(* IEC 61131-3 sources: F100R_S278_Temperville/MyController.device.xml.v3^/Plc Logic.plclogic.xml.v3^/Application.application.xml.v3^/02_Operação (part 2) *)

(* ---- H_MesaResfriador.prg.st ---- *)
PROGRAM H_MesaResfriador
VAR
	///Passo da Execução da Movimentação do Resfriador
	PassoMesaResfriador: INT;
	PassoPauseResfriador: INT;
	PassoAlmMesaResfriador: INT;
	PassoManualResfriador: INT;
	///Blocos Nativos
	TpSairResfriamento: TP;
	TpSomDescarga: TP;
	TonMotorSaidaOff: TON;
	///Bloco Conta Tempo de Permanecia no Resfriador
	TempoResfriamento: Temporizador;
	///Bloco Calcula Posições de Paradas da Carga
	CalculosMesaResfriador: CalculosResfriador;
	///Bloco Converte Milimetro em Pulsos
	ConversorMilimPul: MmConversorPulso;
	///Bloco Converte Pulsos em Milimetros
	ConversorPulMilim: PulsoConversorMm;
	///Bloco Seleciona Pulsos para Vidro Fino ou Grosso
	SelecaoPulsos: BlocoSelecaoEspessura;
	iVelocidadeMesaResfriador: INT;
	///Variaveis que Habilitam o Inicio do Ciclo de Resfriamento
	///Variáveis Booleanas Auxiliares
	xFimTempoResfriamento: BOOL;
	xFinalizaVaivemResfriador: BOOL;
	///Variáveis inteiras Auxiliares
	dValEncoVelMinResfriador: DINT;
	dValEncoCargaResfriador: DINT;
	dValEncoAvancoResfriador: DINT;
	dValEncoRecuoResfriador: DINT;
	dValEncoDescargaResfriador: DINT;
	iValorCargaResfriador: INT;
	iValorOscilacaoResfriador: INT;
	iValorDescargaResfriador: INT;
	iTamanhoAreaUtilResfriador: INT;
	iValMilimetroVelMinResfriador: INT;
	iValMilimetroCargaResfriador: INT;
	iValMilimetroAvancoResfriador: INT;
	iValMilimetroRecuoResfriador: INT;
	iValMilimetroDescargaResfriador: INT;
	dTamanhoCargaResfriador: DINT;
	xSairResfriamento: BOOL;
	xSairFornoResfriamento: BOOL;
	xAlarmeTempoMotorSaida: BOOL;
	xDesablePausaMesaResfriamento: BOOL;
END_VAR

// Direcao de Rotação da Mesa do Resfriamento

xAvancandMesaResfriador:=NOT xMotorMesaResfriadorDirecao AND xMotorResfriadorLigado;
xRecuandoMesaResfriador:=xMotorMesaResfriadorDirecao AND xMotorResfriadorLigado;

//SELEÇÃO DOS PARAMETROS PELA ESPESSURA DO VIDRO
SelecaoPulsos(
	xSelecao:= xEspessuraVidroFinoResfriador,
	iEntrada0101:= iValorCargaResfriadorVidroFin,
	iEntrada0102:= iValorCargaResfriadorVidroGro,
	iEntrada0201:= iValorOscilacaoResfriadorVidroFin,
	iEntrada0202:= iValorOscilacaoResfriadorVidroGro,
	iEntrada0301:= iValorDescargaResfriadorVidroFin,
	iEntrada0302:= iValorDescargaResfriadorVidroGro,
	iEntrada0401:= iTamanhoAreaUtilResfriadorVidroFin,
	iEntrada0402:= iTamanhoAreaUtilResfriadorVidroGro,
	iSaida01=> iValorCargaResfriador,
	iSaida02=> iValorOscilacaoResfriador,
	iSaida03=> iValorDescargaResfriador,
	iSaida04=> iTamanhoAreaUtilResfriador);

// CALCULOS DE POSICIONAMENTO
IF iVelocidadeDescargaMesadoForno>4500 THEN
	iValorVelMinimaResfriador:=550;
ELSE
	iValorVelMinimaResfriador:=350;
END_IF

CalculosMesaResfriador(
	DistanciaVelMinResfriador:= iValorVelMinimaResfriador,
	DistanciaCargaResfriador:= iValorCargaResfriador,
	DistanciaOscilacaoResfriador:= iValorOscilacaoResfriador,
	DistanciaDescargaResfriador:= iValorDescargaResfriador,
	TamanhoAreaUtil:=iTamanhoAreaUtilResfriador,///////
	TamanhoCarga:=iTamanhoCargaAtualResfriador,///////
	SetPointVelMinCarga=> iValMilimetroVelMinResfriador,
	SetPointCargaResfriador=> iValMilimetroCargaResfriador,
	SetPointDescargaResfriador=> iValMilimetroDescargaResfriador,
	SetPointAvancaVaiVemResfriador=> iValMilimetroAvancoResfriador,
	SetPointRecuaVaiVemResfriador=> iValMilimetroRecuoResfriador);

// CONVERSÃO MILIMETROS EM PULSOS

ConversorMilimPul(
	dPulso:= 111325,
	dMilimetro:= 6100,
	iEntrMilimetro01:= iValMilimetroVelMinResfriador,
	iEntrMilimetro02:= iValMilimetroCargaResfriador,
	iEntrMilimetro03:= iValMilimetroDescargaResfriador,
	iEntrMilimetro04:= iValMilimetroAvancoResfriador,
	iEntrMilimetro05:= iValMilimetroRecuoResfriador,
	iEntrMilimetro06:= iTamanhoCargaAtualResfriador,
	dSaidaPulso01=> dValEncoVelMinResfriador,
	dSaidaPulso02=> dValEncoCargaResfriador,
	dSaidaPulso03=> dValEncoDescargaResfriador,
	dSaidaPulso04=> dValEncoAvancoResfriador,
	dSaidaPulso05=> dValEncoRecuoResfriador,
	dSaidaPulso06=> dTamanhoCargaResfriador);

// Velovidade do Vai Vem;

iVelocidadeVaiVemMesaResfriador:=iVelocidadeVaiVemResfriador/10;//////////////////////////////

// MOVIMENTAÇÃO DA MESA DO RESFRIADOR
CASE PassoMesaResfriador OF

		0:	IF xLigaCargaResfriador THEN
				PassoMesaResfriador:=1;
			END_IF

		1:	xMesaResfriadorOn:=TRUE;
			xDesablePausaMesaResfriamento:=TRUE;
			IF xPause THEN
				PassoPauseResfriador:=1;
				PassoMesaResfriador:=300;
				xLigaCargaResfriador:=TRUE;
			ELSIF xAlarmeMotorResfriador THEN
				PassoAlmMesaResfriador:=1;
				PassoMesaResfriador:=400;
			ELSE
				PassoMesaResfriador:=2;
			END_IF

		2:	//xIniciaCargaResfriador:=FALSE;
			iVelocidadeMesaResfriador:= iVelocidadeCargaMesaResfriador;(*Velocidade Carga Resfriador*)
			PassoMesaResfriador:=3;

		3: 	xHomeEncoderResfriador:=TRUE;
			PassoMesaResfriador:=7;

		7:	xAvancoMesaResfriador:=TRUE;
			PassoMesaResfriador:=9;

		9:	xHomeEncoderResfriador:=FALSE;
			PassoMesaResfriador:=10;

		10:	xLigaCargaResfriador:=FALSE;
			IF xIniciaCargaResfriador THEN
				PassoMesaResfriador:=11;
			END_IF
			IF xPause THEN
				PassoPauseResfriador:=1;
				PassoMesaResfriador:=300;
				xLigaCargaResfriador:=TRUE;
			END_IF
			IF xAlarmeMotorResfriador THEN
				PassoAlmMesaResfriador:=1;
				PassoMesaResfriador:=400;
			END_IF

		11:	xHomeEncoderResfriador:=TRUE;
			PassoMesaResfriador:=12;

		12:PassoMesaResfriador:=13;

		13:xHomeEncoderResfriador:=FALSE;
			PassoMesaResfriador:=20;

		20:	xIniciaCargaResfriador:=FALSE;
			xCarregandoResfriador:=TRUE;
			xResfriadorEmCiclo:=TRUE;
			iTamanhoCargaAtualResfriador:=iTamanhoCargaAtualForno;
			PassoMesaResfriador:=23;

		21:	xAvancoMesaResfriador:=TRUE;
			PassoMesaResfriador:=23;

		23:	IF (dValorEncoderResfriador>=dValEncoVelMinResfriador) THEN
				PassoMesaResfriador:=29;
			END_IF
			(*IF xCancelaCargaResfriamento THEN
				PassoMesaResfriador:=25;
			END_IF*)
			IF xPause THEN
				PassoPauseResfriador:=21;
				PassoMesaResfriador:=300;
			END_IF
			IF xAlarmeMotorResfriador OR xAlarmeMotorForno OR xAlarmeGeralEncoderMeResfriador OR xAlarmePortaSaidaFornoAberta THEN
				PassoAlmMesaResfriador:=21;
				PassoMesaResfriador:=400;
			END_IF

		25:	xCancelaCargaResfriamento:=FALSE;
			xCarregandoResfriador:=FALSE;
			xResfriadorEmCiclo:=FALSE;
			PassoMesaResfriador:=10;

		28:	xAvancoMesaResfriador:=TRUE;
			PassoMesaResfriador:=29;

		29:	iVelocidadeMesaResfriador:= iVelMinCargaResfriador;(*Velocidade Minima Carga Resfriador*)
			PassoMesaResfriador:=30;

		30: PassoMesaResfriador:=40;
			xDesligaVentilador01	:=TRUE;	//-> TASK/M_Ventilador01 - (*Alterado Tempera de passagem *)
			xFimDescargaMesaPass:=TRUE;

		40: IF (dValorEncoderResfriador>=dValEncoCargaResfriador) THEN
				PassoMesaResfriador:=50;
			END_IF
			IF xPause THEN
				PassoPauseResfriador:=28;
				PassoMesaResfriador:=300;
			END_IF
			IF xAlarmeMotorResfriador OR xAlarmeGeralEncoderMeResfriador THEN
				PassoAlmMesaResfriador:=28;
				PassoMesaResfriador:=400;
			END_IF

		50: xCarregandoResfriador:=FALSE;
			xResfriadorCarregado:= TRUE;
			xResfriadorCheio:=TRUE;
			xInicioPrimeiroEstagio:=TRUE;
			xReajustaAlturaDuctosInf01:=TRUE;(* Alterado para tempera de passagem *)
			xReajustaAlturaDuctosSup01:=TRUE;(* Alterado para tempera de passagem *)
			//xDesligaVentilador01	:=TRUE;	//-> TASK/M_Ventilador01 - (*Alterado Tempera de passagem *)
			xDesligaVentilador02	:=TRUE;	//-> TASK/M_Ventilador02 - (*Alterado Tempera de passagem *)
			xFechVenezVentPass		:=TRUE; //-> TASK/T_VenezianaVentInfPass
			PassoMesaResfriador:=55;

		55: xAvancoMesaResfriador:=FALSE;
			PassoMesaResfriador:=60;

		60:	iVelocidadeMesaResfriador:= 1*iVelocidadeVaiVemMesaResfriador;(*-Velocidade VaiVem Resfriador*)
			PassoMesaResfriador:=61;

		61:	xRecuoMesaResfriador:=TRUE;
			PassoMesaResfriador:=62;

		62:	xDesablePausaMesaResfriamento:=FALSE;
			PassoMesaResfriador:=70;

		70: IF NOT xFinalizaVaivemResfriador THEN
				IF (dValorEncoderResfriador<=dValEncoRecuoResfriador) THEN
					PassoMesaResfriador:=80;
				END_IF
				IF iVelocidadeMesaResfriador <> 1*iVelocidadeVaiVemMesaResfriador THEN
					PassoMesaResfriador:=60;
				END_IF
				IF xPause THEN
					PassoPauseResfriador:=60;
					PassoMesaResfriador:=300;
				END_IF
				IF xAlarmeMotorResfriador OR xAlarmeGeralEncoderMeResfriador THEN
					PassoAlmMesaResfriador:=60;
					PassoMesaResfriador:=400;
				END_IF
			ELSE
				xPausaMesaResfrimento:=FALSE;
				xDesablePausaMesaResfriamento:=TRUE;
				PassoMesaResfriador:=115;
			END_IF

		80:	xRecuoMesaResfriador:=FALSE;
			PassoMesaResfriador:=90;

		90:iVelocidadeMesaResfriador:= iVelocidadeVaiVemMesaResfriador;(*-Velocidade VaiVem Resfriador*)
			PassoMesaResfriador:=91;

		91:	xAvancoMesaResfriador:=TRUE;
			PassoMesaResfriador:=100;

		100:PassoMesaResfriador:=101;

		101:IF NOT xFinalizaVaivemResfriador THEN
				IF (dValorEncoderResfriador>=dValEncoAvancoResfriador) THEN
					PassoMesaResfriador:=110;
				END_IF
				IF iVelocidadeMesaResfriador <> iVelocidadeVaiVemMesaResfriador THEN
					PassoMesaResfriador:=90;
				END_IF
				IF xPause THEN
					PassoPauseResfriador:=90;
					PassoMesaResfriador:=300;
				END_IF
				IF xAlarmeMotorResfriador OR xAlarmeGeralEncoderMeResfriador THEN
					PassoAlmMesaResfriador:=90;
					PassoMesaResfriador:=400;
				END_IF
			ELSE
				xPausaMesaResfrimento:=FALSE;
				xDesablePausaMesaResfriamento:=TRUE;
				PassoMesaResfriador:=120;
			END_IF

		110: xAvancoMesaResfriador:=FALSE;
			 PassoMesaResfriador:=60;

		115:xRecuoMesaResfriador:=FALSE;
			PassoMesaResfriador:=116;

		116:xAvancoMesaResfriador:=TRUE;
			PassoMesaResfriador:=120;

		120:PassoMesaResfriador:=130;

		130:iVelocidadeMesaResfriador:= iVelocidadeDescargaMesaResfriador;(*-Velocidade Descarga Resfriador*)
			PassoMesaResfriador:=140;

		140: IF xDescarregandoResfriador THEN
				 PassoMesaResfriador:=150;
			 ELSE
				 PassoMesaResfriador:=141;
			 END_IF

		141:xDescarregandoResfriador:=TRUE;
			xInicioDescargaMesaSaida:=TRUE;
			//xDesligaVentilador01		:=TRUE;	//-> TASK/M_Ventilador01 - (*Alterado Tempera de passagem *)
			//xDesligaVentilador02		:=TRUE;	//-> TASK/M_Ventilador02 - (*Alterado Tempera de passagem *)
			xDesligaVentilador03		:=TRUE;	//-> TASK/M_Ventilador03
			//xDesligaVentilador04		:=TRUE;	//-> TASK/M_Ventilador04
			xFimTrocaEstagiosResfriador:=TRUE; //-> TASK/EstagiosResfriador
			xDesceGradeMesaSaida:=TRUE;
			xReajustaAlturaDuctosSup02:=TRUE;; // ->TASK/J_DuctosResfriadorSup02
			xResfriadorCarregado:= FALSE;
			xFimTempoResfriamento:=FALSE;
			xFinalizaVaivemResfriador:=FALSE;
			iContaCargasResfriamento:=iContaCargasResfriamento+1;
			PassoMesaResfriador:=150;

		150:IF (dValorEncoderResfriador>=dValEncoDescargaResfriador) THEN
				PassoMesaResfriador:=155;
			END_IF
			IF xPause THEN
				PassoPauseResfriador:=130;
				PassoMesaResfriador:=300;
			END_IF
			IF xAlarmeMotorResfriador OR xAlarmeMotorSaida (*xAlarmeTempoMotorSaida*) OR xAlarmeGeralEncoderMeResfriador THEN
				PassoAlmMesaResfriador:=130;
				PassoMesaResfriador:=400;
			END_IF

		155: xFimDescargaMesaSaida:=TRUE;  //->TASK/MesaSaida
			 PassoMesaResfriador:=156;

		156: xAvancoMesaResfriador:=FALSE;
			 PassoMesaResfriador:=160;

		160:xDescarregandoResfriador:=FALSE;
			xMesaResfriadorOn:=FALSE;
			xResfriadorEmCiclo:=FALSE;
			xDesabJogMesaSaida:=FALSE;//->TASK/MesaSaida
			//xFimDescargaMesaSaida:=TRUE;  //->TASK/MesaSaida
			//xFimTrocaEstagiosResfriador:=TRUE; //-> TASK/EstagiosResfriador
			xResfriadorCheio:=FALSE;
			iTamanhoCargaAtualResfriador:=0;
			PassoMesaResfriador:=170;

		170://xReajustaAlturaDuctosInf01:=TRUE;
			//xReajustaAlturaDuctosSup01:=TRUE;
			xReajustaAlturaDuctosInf02:=TRUE;
			//xReajustaAlturaDuctosSup02:=TRUE;
			xDesablePausaMesaResfriamento:=FALSE;
			PassoMesaResfriador:=0;

		// Emergência Pausa/Reinicio
		300:xAvancoMesaResfriador:=FALSE;
			xRecuoMesaResfriador:=FALSE;
			PassoMesaResfriador:=301;

		301:PassoMesaResfriador:=302;

		302:IF xRestart THEN
				PassoMesaResfriador:=303;
			END_IF

		303:PassoMesaResfriador:=PassoPauseResfriador;

		// Alarme Motor Parada/Reinicio
	400:xAvancoMesaResfriador:=FALSE;
		xRecuoMesaResfriador:=FALSE;
		PassoMesaResfriador:=401;

	401:PassoMesaResfriador:=402;

	402:IF (xRestart) AND iCanOpenInverMesaResfrStateOk  THEN
			PassoMesaResfriador:=PassoAlmMesaResfriador;
		END_IF
END_CASE

//Comando Sair forno foi acionado com carga no Resfriamento
IF xResfriadorCarregado AND xSairForno THEN
	xSairFornoResfriamento:=TRUE;
END_IF

TpSairResfriamento(IN:=xBtSairResfriamento OR xSairFornoResfriamento , PT:=T#500MS , Q=>xSairResfriamento , ET=> );
IF xBtSairResfriamento THEN
	xBtSairResfriamento:=FALSE;
	xSairResfriamentoEventos:=TRUE;
END_IF
IF xSairFornoResfriamento THEN
	xSairFornoResfriamento:=FALSE;
END_IF

// TEMPORIZADORES

TempoResfriamento(
	IniciaTempo:= xResfriadorCarregado,
	AbortaTempo:= xSairResfriamento OR xOperacaoManual,
	SetPointTempo:= iTempoResfriamento,
	FimTempo:= 		xFimTempoResfriamento,
	TempoDecorrido=>iTempoResfriamentoDecorrido,
	TempoRestante=> iTempoResfriamentoRestante);

xFinalizaVaivemResfriador:=xFimTempoResfriamento;

TpSomDescarga(IN:= xFimTempoResfriamento, PT:=T#5S , Q=>xSomDescarga , ET=> );

IF (iTempoResfriamentoRestante <= 2) and xResfriadorCheio THEN
	xDesabJogMesaSaida:=TRUE;//->TASK/MesaSaida
END_IF

//STATUS
xResfriadorVazio:=NOT xResfriadorCheio;

xPausaResfrChAbreSupAcionanda:=(xPausaMesaResfrimento AND NOT xDesablePausaMesaResfriamento);
// MOVIMENTAÇÃO PELO COMANDO ENTRADAS DIGITAIS DO INVERSOR
// Comando e Direção
xMotorMesaResfriadorAvanco:= xAvancoMesaResfriador;// AND NOT (xPausaResfrChAbreSupAcionanda);
xMotorMesaResfriadorRecuo:= xRecuoMesaResfriador;// AND NOT (xPausaResfrChAbreSupAcionanda);

InversorMesaResfri.i_xAvanco:=xMotorMesaResfriadorAvanco;
InversorMesaResfri.i_xRecuo:=xMotorMesaResfriadorRecuo;

// Velocidade
InversorMesaResfri.i_iFreqRef:=iVelocidadeMesaResfriador;

//---------------------------------------------------------------------------------\\

IF xOperacaoManual THEN
	PassoMesaResfriador:=0;
	PassoPauseResfriador:=0;
	PassoAlmMesaResfriador:=0;
	xLigaCargaResfriador:=FALSE;
	xIniciaCargaResfriador:=FALSE;
	xCarregandoResfriador:=FALSE;
	xMesaResfriadorOn:=FALSE;
	xResfriadorEmCiclo:=FALSE;
	xCancelaCargaResfriamento:=FALSE;
	xResfriadorCarregado:= FALSE;
	xDescarregandoResfriador:=FALSE;
	xInicioDescargaMesaSaida:=FALSE;
	xFimTempoResfriamento:=FALSE;
	xFinalizaVaivemResfriador:=FALSE;
	xFimTempoResfriamento:=FALSE;
	xBtSairResfriamento:=FALSE;
	xSairFornoResfriamento:=FALSE;
	xPulsoTrocaParamResfriador:=FALSE;
	xResfriadorCheio:=FALSE;
	iTamanhoCargaAtualResfriador:=0;
	xDesabJogMesaSaida:=FALSE;
	xFechVenezVentPass		:=FALSE;

	xAvancoMesaResfriador:=FALSE;
	xRecuoMesaResfriador:=FALSE;
	xDesablePausaMesaResfriamento:=FALSE;
END_IF

IF	uHoraRealTime=0 AND uMinutoRealTime=0 AND uSegundoRealTime=0 THEN
	iContaCargasResfriamento:=0;
END_IF

// Tempo para ligar Motor da Saida ou gerar Alarme
TonMotorSaidaOff(IN:=xInicioDescargaMesaSaida AND NOT xMotorSaidaLigado, PT:= T#300MS , Q=> xAlarmeTempoMotorSaida , ET=> );

(* ---- I_MesaSaida.prg.st ---- *)
PROGRAM I_MesaSaida
VAR
	PassoMesaSaida: INT;
	PassoPauseSaida: INT;
	PassoAlmSaida: INT;
	PassoManualSaida: INT;
	///Blocos Nativos
	///Blocos Criados
	PulsoPoChAvanco: PulsoPositivo;
	PulsoNeChAvanco: PulsoNegativo;
	PulsoPoSensorDesl: PulsoPositivo;
	xAvancoMesaSaida: BOOL;
	xRecuoMesaSaida: BOOL;
	xAvancoJogMesaSaida: BOOL;
	xRecuoJogMesaSaida: BOOL;
	xChAvancaMesaSaidaPo: BOOL;
	xChAvancaMesaSaidaNe: BOOL;
	xSensorDesligaMesaSaidaPo: BOOL;
	iVelocidadeMesaSaida: INT;
END_VAR

// JOG DA MESA DE SAIDA
(*Avanço*)
PulsoPoChAvanco(Entrada:= xChAvancaMesaSaida, SaidaPulsoPo=>xChAvancaMesaSaidaPo );
PulsoNeChAvanco(Entrada:= xChAvancaMesaSaida, SaidaPulsoNe=>xChAvancaMesaSaidaNe );
PulsoPoSensorDesl(Entrada:= xSensorDesligaMesaSaida, SaidaPulsoPo=>xSensorDesligaMesaSaidaPo );

IF xChAvancaMesaSaidaPo AND NOT xDescarregandoResfriador AND NOT xDesabJogMesaSaida (*AND NOT xPausaEmergencia*) THEN
	xAvancoJogMesaSaida:=TRUE;
END_IF
IF xChRecuaMesaSaida OR xSensorDesligaMesaSaidaPo THEN
	xAvancoJogMesaSaida:=FALSE;
END_IF

(*Recuo*)
IF xChRecuaMesaSaida AND NOT xDescarregandoResfriador AND NOT xDesabJogMesaSaida  (*AND NOT xPausaEmergencia*) THEN
	xRecuoJogMesaSaida:=TRUE;
ELSE
	xRecuoJogMesaSaida:=FALSE;
END_IF

// SEQUENCIA DE DESCARREGAMENTO

CASE PassoMesaSaida OF

		0:	IF xInicioDescargaMesaSaida THEN
				PassoMesaSaida:=1;
			END_IF

		1:	IF xPause THEN
				PassoPauseSaida:=0;
				PassoMesaSaida:=300;
			ELSIF xAlarmeMotorSaida THEN
				PassoAlmSaida:=0;
				PassoMesaSaida:=400;
			ELSE
				PassoMesaSaida:=2;
			END_IF

		2:	iVelocidadeMesaSaida:= iVelociadeCargaMesadeSaida;(*Velocidade Descarga Mesa Saida*)
			PassoMesaSaida:=5;

		5: xAvancoMesaSaida:=TRUE;
			PassoMesaSaida:=10;

		10:	xInicioDescargaMesaSaida:=FALSE;
			PassoMesaSaida:=20;

		20:	IF xFimDescargaMesaSaida THEN
				PassoMesaSaida:=25;
			END_IF
			IF xPause THEN
				PassoPauseSaida:=2;
				PassoMesaSaida:=300;
			END_IF
			IF xAlarmeMotorSaida OR xAlarmeMotorResfriador OR xAlarmeGeralEncoderMeResfriador THEN
				PassoAlmSaida:=2;
				PassoMesaSaida:=400;
			END_IF

		25:	xAvancoMesaSaida:=FALSE;
			PassoMesaSaida:=30;

		30:	xFimDescargaMesaSaida:=FALSE;
			PassoMesaSaida:=0;

		// Emergência Pausa/Reinicio
		300:xAvancoMesaSaida:=FALSE;
			PassoMesaSaida:=301;

		301:PassoMesaSaida:=302;

		302:IF xRestart THEN
				PassoMesaSaida:=303;
			END_IF

		303: PassoMesaSaida:=PassoPauseSaida;

		// Alarme Motor Parada/Reinicio
		400:xAvancoMesaSaida:=FALSE;
			PassoMesaSaida:=401;

		401:PassoMesaSaida:=402;

		402:IF xRestart AND iCanOpenInverMesaSaidaStateOk THEN
				PassoMesaSaida:=PassoAlmSaida;
			END_IF

END_CASE

// MOVIMENTAÇÃO PELO COMANDO ENTRADAS DIGITAIS DO INVERSOR
// Comando e Direção
xMotorMesaSaidaAvanco:= xAvancoMesaSaida OR xAvancoJogMesaSaida;
xMotorMesaSaidaRecuo:= xRecuoMesaSaida OR xRecuoJogMesaSaida;

InversorMesaSaida.i_xAvanco:=xMotorMesaSaidaAvanco;
InversorMesaSaida.i_xRecuo:=xMotorMesaSaidaRecuo;

// Velocidade
IF xAvancoJogMesaSaida OR xRecuoJogMesaSaida THEN
	InversorMesaSaida.i_iFreqRef:=iVelocidadeJogMesaSaida;
ELSE
	InversorMesaSaida.i_iFreqRef:=iVelocidadeMesaSaida;
END_IF
//--------------------------------------------------------------------------\\

IF xOperacaoManual THEN
	PassoMesaSaida:=0;
	xInicioDescargaMesaSaida:=FALSE;
	xFimDescargaMesaSaida:=FALSE;
	xAvancoMesaSaida:=FALSE;
	xRecuoMesaSaida:=FALSE;
	xAvancoJogMesaSaida:=FALSE;
	xRecuoJogMesaSaida:=FALSE;
END_IF

(* ---- J_DuctosResfriadorInf01.prg.st ---- *)
PROGRAM J_DuctosResfriadorInf01
VAR
	PassoHomeDuctosResfrInf01: INT;
	PassoPausaHomeDuctosResfrInf01: INT;
	PassoAlmHomeDuctosResfrInf01: INT;
	PassoAjusteDuctosResfInf01: INT;
	PassoPausaAjusteDuctosResfInf01: INT;
	PassoAlmAjusteDuctosResfInf01: INT;
	PassoChaveDuctosResfrInf01: INT;
	PassoPausaChaveDuctosResfrInf01: INT;
	PassoAlmChaveDuctosResfrInf01: INT;
	/// Bloco Movimenta Ductos do Resfriador
	McMoveVelocityDuctosInf01: GIPLC.MC_MoveVelocity;
	/// Bloco Desliga Motor Ductos do Resfriador
	McStopDuctosResfriadorInf01: GIPLC.MC_Stop;
	/// Bloco Jog Motor Ductos do Resfriador
	McJogDuctosResfriadorInf01: GIPLC.MC_Jog;
	///Bloco Converte Milimetro em Pulsos
	ConversorMilimPul01ResfrInf01: MmConversorPulso;
	///Bloco Converte Milimetro em Pulsos
	ConversorMilimPul02ResfrInf01: MmConversorPulso;
	///Bloco Converte Pulsos em Milimetros
	ConversorPulMilimResfrInf01: PulsoConversorMm;
	xExecutaMovDuctosResfriadorInf01: BOOL;
	xExecutaStopDuctosResfriadorInf01: BOOL;
	xStopMesaDuctosResfriadorInf01Done: BOOL;
	xAbreDuctosResfriadorInf01: BOOL;
	xFechaDuctosResfriadorInf01: BOOL;
	xAjustarAlturaResfriadorInf01: BOOL;
	///Recebera uma valor fixo
	iVelocidadeHomeDuctosResfrInf01: INT;
	iVelocidadeJogDuctosResfrInf01: INT;
	iVelocidadeDuctosResfriadorInf01: INT;
	dValEncoAltura01ResfriadorInf01: DINT;
	dValEncoAltura02ResfriadorInf01: DINT;
	dValEncoAltura03ResfriadorInf01: DINT;
	dValEncoAlturaResfriadorInf01: DINT;
	dValEncoToleranciaResfrInf01: DINT;
	dValEncoAlturaVelMinimaResfrInf01: DINT := 35;
	xDifusorInf01Fechando: BOOL;
	xDifusorInf01Abrindo: BOOL;
	iCompValAltura01ResfriadorInf01: INT;
	iCompValAltura02ResfriadorInf01: INT;
	iCompValAltura03ResfriadorInf01: INT;
	iCompAlturaAtualDuctosResfriadorInf01: INT;
	iCompessaAlturaDuctosResfriadorInf01: INT;
END_VAR

iCompessaAlturaDuctosResfriadorInf01:=REAL_TO_INT(rOffSetResfInf01);
iCompValAltura01ResfriadorInf01:=	iValAltura01ResfriadorInf01 - iCompessaAlturaDuctosResfriadorInf01;
iCompValAltura02ResfriadorInf01:=	iValAltura02ResfriadorInf01 - iCompessaAlturaDuctosResfriadorInf01;
iCompValAltura03ResfriadorInf01:=	iValAltura03ResfriadorInf01 - iCompessaAlturaDuctosResfriadorInf01;

// CONVERSÃO MILIMETROS EM PULSOS
ConversorMilimPul01ResfrInf01(
	dPulso:= 1261,
	dMilimetro:= 133,
	iEntrMilimetro01:= iCompValAltura01ResfriadorInf01,
	iEntrMilimetro02:= iCompValAltura02ResfriadorInf01,
	iEntrMilimetro03:= iCompValAltura03ResfriadorInf01,
	dSaidaPulso01=> dValEncoAltura01ResfriadorInf01,
	dSaidaPulso02=> dValEncoAltura02ResfriadorInf01,
	dSaidaPulso03=> dValEncoAltura03ResfriadorInf01);

ConversorMilimPul02ResfrInf01(
	dPulso:= 1261,
	dMilimetro:= 133,
	iEntrMilimetro01:= 2,//iValEncoToleranciaDuctosInf01,
	iEntrMilimetro02:= 8,//iValEncoAlturaVelMinimaDuctosInf01,
	dSaidaPulso01=> dValEncoToleranciaResfrInf01,
	dSaidaPulso02=> dValEncoAlturaVelMinimaResfrInf01);

// SEQUENCIA DE HOME

CASE PassoHomeDuctosResfrInf01 OF

		0:	IF xIniciaHomeDuctosInf01 THEN
				PassoHomeDuctosResfrInf01:=5;
			END_IF

		5:	IF xChAbreDuctosResfriadorInf01 THEN
				PassoHomeDuctosResfrInf01:=6;
			ELSE
				PassoHomeDuctosResfrInf01:=10;
			END_IF

		6:	xIniciaHomeDuctosInf01:=FALSE;
			PassoHomeDuctosResfrInf01:=0;

		10:	xIniciaHomeDuctosInf01:=FALSE;
			xHomeDuctosResfriadorInf01Ok:=FALSE;
			xAjusteAlturaDuctosInf01OK:=FALSE;
			xDuctosInf01EmHome:=TRUE;
			iVelocidadeDuctosResfriadorInf01:= -150;//1*iVelocidadeHomeDuctosResfrInf01;
			xExecutaMovDuctosResfriadorInf01:=TRUE;
			IF McMoveVelocityDuctosInf01.Busy THEN
				PassoHomeDuctosResfrInf01:=20;
			END_IF

		20:	xExecutaMovDuctosResfriadorInf01:=FALSE;
			IF xSensorFechadoResfriadorInf01 THEN
				PassoHomeDuctosResfrInf01:=50;
			END_IF
			IF xPause THEN
				PassoPausaHomeDuctosResfrInf01:=10;
				PassoHomeDuctosResfrInf01:=300;
			END_IF
			IF xAlarmeMotorDifusorInf01 THEN
				PassoAlmHomeDuctosResfrInf01:=10;
				PassoHomeDuctosResfrInf01:=400;
			END_IF

		(*30: xExecutaStopDuctosResfriadorInf01:=TRUE;
			IF	xStopMesaDuctosResfriadorInf01Done THEN
				PassoHomeDuctosResfrInf01:=40;
			END_IF

		40: xExecutaStopDuctosResfriadorInf01:=FALSE;
			PassoHomeDuctosResfrInf01:=50;*)

		50:	iVelocidadeDuctosResfriadorInf01:= 50;
			xExecutaMovDuctosResfriadorInf01:=TRUE;
			IF McMoveVelocityDuctosInf01.Busy THEN
				PassoHomeDuctosResfrInf01:=60;
			END_IF

		60:	xExecutaMovDuctosResfriadorInf01:=FALSE;
			IF NOT xSensorFechadoResfriadorInf01 THEN
				PassoHomeDuctosResfrInf01:=70;
			END_IF
			IF xPause THEN
				PassoPausaHomeDuctosResfrInf01:=50;
				PassoHomeDuctosResfrInf01:=300;
			END_IF
			IF xAlarmeMotorDifusorInf01 THEN
				PassoAlmHomeDuctosResfrInf01:=50;
				PassoHomeDuctosResfrInf01:=400;
			END_IF

		70:	xExecutaStopDuctosResfriadorInf01:=TRUE;
			IF	xStopMesaDuctosResfriadorInf01Done THEN
				xHomeEncoderDuctosResfriadorInf01:=TRUE;
				PassoHomeDuctosResfrInf01:=80;
			END_IF

		80: xHomeEncoderDuctosResfriadorInf01:=FALSE;
			xExecutaStopDuctosResfriadorInf01:=FALSE;
			xDuctosInf01EmHome:=FALSE;
			xHomeDuctosResfriadorInf01Ok:=TRUE;

		// Emergência Pausa/Reinicio
		300:xExecutaStopDuctosResfriadorInf01:=TRUE;
			PassoHomeDuctosResfrInf01:=301;

		301:xExecutaStopDuctosResfriadorInf01:=FALSE;
			xExecutaMovDuctosResfriadorInf01:=FALSE;
			xDuctosInf01EmHome:=FALSE;
			PassoHomeDuctosResfrInf01:=302;

		302:IF xRestart THEN
				PassoHomeDuctosResfrInf01:=303;
			END_IF

		303:IF xInvDuctosInf01Habilitado THEN
				PassoHomeDuctosResfrInf01:=0;//PassoPausaHomeDuctosResfrInf01;
			END_IF

		// Alarme Motor Parada/Reinicio
		400:xExecutaStopDuctosResfriadorInf01:=TRUE;
			PassoHomeDuctosResfrInf01:=401;

		401:xExecutaStopDuctosResfriadorInf01:=FALSE;
			xExecutaMovDuctosResfriadorInf01:=FALSE;
			PassoHomeDuctosResfrInf01:=402;

		402:IF xRestart AND xInvDuctosInf01Habilitado THEN
				PassoHomeDuctosResfrInf01:=PassoAlmHomeDuctosResfrInf01;
			END_IF
END_CASE

//
//IF xTerceiroEstagioResfriador THEN
//	dValEncoAlturaResfriadorInf01:=dValEncoAltura03ResfriadorInf01;
//ELSIF xSegundoEstagioResfriador THEN
//	dValEncoAlturaResfriadorInf01:=dValEncoAltura02ResfriadorInf01;
//ELSE
	dValEncoAlturaResfriadorInf01:=dValEncoAltura01ResfriadorInf01;
//END_IF

// SEQUENCIA DE FUNCIONAMENTO

IF (xBtRecAjustaAlturaDuctosInf01 OR BtParamDuctosResfriadorInf01 OR xLigaSegEstagDuctosInf01 OR xLigaTerEstagDuctosInf01 OR xReajustaAlturaDuctosInf01) AND xHomeDuctosResfriadorInf01Ok THEN
	xAjustarAlturaResfriadorInf01:=TRUE;
	xBtRecAjustaAlturaDuctosInf01:=FALSE;
	BtParamDuctosResfriadorInf01:=FALSE;
	xLigaSegEstagDuctosInf01:= FALSE;
	xLigaTerEstagDuctosInf01:= FALSE;
	xReajustaAlturaDuctosInf01:=FALSE;
ELSE
	xBtRecAjustaAlturaDuctosInf01:=FALSE;
	BtParamDuctosResfriadorInf01:=FALSE;
	xLigaSegEstagDuctosInf01:= FALSE;
	xLigaTerEstagDuctosInf01:= FALSE;
	xReajustaAlturaDuctosInf01:=FALSE;
END_IF

CASE PassoAjusteDuctosResfInf01 OF

		0:	IF xAjustarAlturaResfriadorInf01 AND NOT xChAbreDuctosResfriadorInf01 THEN
				PassoAjusteDuctosResfInf01:=10;
			END_IF

		10:	xAjustarAlturaResfriadorInf01:=FALSE;
			xAjusteAlturaDuctosInf01OK:=FALSE;
			xDuctosInf01EmAjuste:=TRUE;
			IF dValorEncoderDuctosResfriadorInf01<dValEncoAlturaResfriadorInf01-dValEncoToleranciaResfrInf01 THEN
				xDifusorInf01Abrindo:=TRUE;
				PassoAjusteDuctosResfInf01:=20;//Sobe
			END_IF
			IF dValorEncoderDuctosResfriadorInf01>dValEncoAlturaResfriadorInf01+dValEncoToleranciaResfrInf01 THEN
				PassoAjusteDuctosResfInf01:=100;//Desce
				xDifusorInf01Fechando:=TRUE;
			END_IF
			IF dValorEncoderDuctosResfriadorInf01>=dValEncoAlturaResfriadorInf01-dValEncoToleranciaResfrInf01 AND dValorEncoderDuctosResfriadorInf01<=dValEncoAlturaResfriadorInf01+dValEncoToleranciaResfrInf01 THEN
				PassoAjusteDuctosResfInf01:=180;//Não se Move
			END_IF
//Sobe
		20:	iVelocidadeDuctosResfriadorInf01:= iVelocidadeAjusteDuctosResfriadorInf01;
			xExecutaMovDuctosResfriadorInf01:=TRUE;
			IF McMoveVelocityDuctosInf01.Busy THEN
				PassoAjusteDuctosResfInf01:=30;
			END_IF

		30:	xExecutaMovDuctosResfriadorInf01:=FALSE;
			IF dValorEncoderDuctosResfriadorInf01>=dValEncoAlturaResfriadorInf01-35(*dValEncoAlturaVelMinimaResfrInf01*) THEN
				PassoAjusteDuctosResfInf01:=40;
			END_IF
			IF iVelocidadeDuctosResfriadorInf01<> iVelocidadeAjusteDuctosResfriadorInf01 THEN
				PassoAjusteDuctosResfInf01:=20;
			END_IF
			IF xPause THEN
				PassoPausaAjusteDuctosResfInf01:=20;
				PassoAjusteDuctosResfInf01:=300;
			END_IF
			IF xAlarmeMotorDifusorInf01 THEN
				PassoAlmAjusteDuctosResfInf01:=20;
				PassoAjusteDuctosResfInf01:=400;
			END_IF

		40:	iVelocidadeDuctosResfriadorInf01:= iVelocidadeMinimaDuctosResfriadorInf01;
			xExecutaMovDuctosResfriadorInf01:=TRUE;
			IF McMoveVelocityDuctosInf01.Busy THEN
				PassoAjusteDuctosResfInf01:=50;
			END_IF

		50:	xExecutaMovDuctosResfriadorInf01:=FALSE;
			IF (dValorEncoderDuctosResfriadorInf01>=dValEncoAlturaResfriadorInf01) OR xSensorAbertoResfriadorInf01 THEN
				PassoAjusteDuctosResfInf01:=60;
			END_IF
			IF xPause THEN
				PassoPausaAjusteDuctosResfInf01:=40;
				PassoAjusteDuctosResfInf01:=300;
			END_IF
			IF xAlarmeMotorDifusorInf01 THEN
				PassoAlmAjusteDuctosResfInf01:=40;
				PassoAjusteDuctosResfInf01:=400;
			END_IF

		60: xExecutaStopDuctosResfriadorInf01:=TRUE;
			IF	xStopMesaDuctosResfriadorInf01Done THEN
				PassoAjusteDuctosResfInf01:=180;
			END_IF
//Desce
		100:iVelocidadeDuctosResfriadorInf01:= -1*iVelocidadeAjusteDuctosResfriadorInf01;
			xExecutaMovDuctosResfriadorInf01:=TRUE;
			IF McMoveVelocityDuctosInf01.Busy THEN
				PassoAjusteDuctosResfInf01:=110;
			END_IF

		110:xExecutaMovDuctosResfriadorInf01:=FALSE;
			IF dValorEncoderDuctosResfriadorInf01 <= dValEncoAlturaResfriadorInf01+35(*dValEncoAlturaVelMinimaResfrInf01*) THEN
				PassoAjusteDuctosResfInf01:=120;
			END_IF
			IF iVelocidadeDuctosResfriadorInf01<> -1*iVelocidadeAjusteDuctosResfriadorInf01 THEN
				PassoAjusteDuctosResfInf01:=100;
			END_IF
			IF xPause THEN
				PassoPausaAjusteDuctosResfInf01:=100;
				PassoAjusteDuctosResfInf01:=300;
			END_IF
			IF xAlarmeMotorDifusorInf01 THEN
				PassoAlmAjusteDuctosResfInf01:=100;
				PassoAjusteDuctosResfInf01:=400;
			END_IF

		120:iVelocidadeDuctosResfriadorInf01:= -1*iVelocidadeMinimaDuctosResfriadorInf01;
			xExecutaMovDuctosResfriadorInf01:=TRUE;
			IF McMoveVelocityDuctosInf01.Busy THEN
				PassoAjusteDuctosResfInf01:=130;
			END_IF

		130:xExecutaMovDuctosResfriadorInf01:=FALSE;
			IF dValorEncoderDuctosResfriadorInf01<=dValEncoAlturaResfriadorInf01 THEN
				PassoAjusteDuctosResfInf01:=140;
			END_IF
			IF xPause THEN
				PassoPausaAjusteDuctosResfInf01:=120;
				PassoAjusteDuctosResfInf01:=300;
			END_IF
			IF xAlarmeMotorDifusorInf01 THEN
				PassoAlmAjusteDuctosResfInf01:=120;
				PassoAjusteDuctosResfInf01:=400;
			END_IF

		140:xExecutaStopDuctosResfriadorInf01:=TRUE;
			IF	xStopMesaDuctosResfriadorInf01Done THEN
				PassoAjusteDuctosResfInf01:=180;
			END_IF
//Fim
		180:xDifusorInf01Abrindo:=FALSE;
			xDifusorInf01Fechando:=FALSE;
			xExecutaStopDuctosResfriadorInf01:=FALSE;
			xDuctosInf01EmAjuste:=FALSE;
			xAjusteAlturaDuctosInf01OK:=TRUE;
			PassoAjusteDuctosResfInf01:=0;

		// Emergência Pausa/Reinicio
		300:xExecutaStopDuctosResfriadorInf01:=TRUE;
			PassoAjusteDuctosResfInf01:=301;

		301:xExecutaStopDuctosResfriadorInf01:=FALSE;
			xExecutaMovDuctosResfriadorInf01:=FALSE;
			PassoAjusteDuctosResfInf01:=302;

		302:IF xRestart THEN
				PassoAjusteDuctosResfInf01:=303;
			END_IF

		303:IF xInvDuctosInf01Habilitado THEN
				PassoAjusteDuctosResfInf01:=PassoPausaAjusteDuctosResfInf01;
			END_IF

		// Alarme Motor Parada/Reinicio
		400:xExecutaStopDuctosResfriadorInf01:=TRUE;
			PassoAjusteDuctosResfInf01:=401;

		401:xExecutaStopDuctosResfriadorInf01:=FALSE;
			xExecutaMovDuctosResfriadorInf01:=FALSE;
			PassoAjusteDuctosResfInf01:=402;

		402:IF xRestart AND xInvDuctosInf01Habilitado THEN
				PassoAjusteDuctosResfInf01:=PassoAlmAjusteDuctosResfInf01;
			END_IF

END_CASE

// MOVIMENTO COM A CHAVE DE ABERTURA

CASE PassoChaveDuctosResfrInf01 OF

		0:	IF xChAbreDuctosResfriadorInf01 AND xHomeDuctosResfriadorInf01Ok THEN
				PassoChaveDuctosResfrInf01:=10;
				PassoAjusteDuctosResfInf01:=0;
			END_IF

		10:	iVelocidadeJogDuctosResfrInf01:=iVelocidadeAjusteDuctosResfriadorInf01;
			xAjusteAlturaDuctosInf01OK:=FALSE;
			xAbreDuctosResfriadorInf01:=xChAbreDuctosResfriadorInf01;
			IF xSensorAbertoResfriadorInf01 THEN
				PassoChaveDuctosResfrInf01:=20;
			END_IF
			IF xPause THEN
				PassoPausaChaveDuctosResfrInf01:=10;
				PassoChaveDuctosResfrInf01:=300;
			END_IF
			IF xAlarmeMotorDifusorInf01 THEN
				PassoAlmChaveDuctosResfrInf01:=10;
				PassoChaveDuctosResfrInf01:=400;
			END_IF

		20:	xAbreDuctosResfriadorInf01:=FALSE;
			PassoChaveDuctosResfrInf01:=21;

		21:	IF NOT xChAbreDuctosResfriadorInf01 THEN
				PassoChaveDuctosResfrInf01:=0;
				PassoAjusteDuctosResfInf01:=100;
			END_IF
			IF xPause THEN
				PassoPausaChaveDuctosResfrInf01:=21;
				PassoChaveDuctosResfrInf01:=300;
			END_IF
			IF xAlarmeMotorDifusorInf01 THEN
				PassoAlmChaveDuctosResfrInf01:=21;
				PassoChaveDuctosResfrInf01:=400;
			END_IF

		// Emergência Pausa/Reinicio
		300:xExecutaStopDuctosResfriadorInf01:=TRUE;
			PassoChaveDuctosResfrInf01:=301;

		301:xExecutaStopDuctosResfriadorInf01:=FALSE;
			xExecutaMovDuctosResfriadorInf01:=FALSE;
			PassoChaveDuctosResfrInf01:=302;

		302:IF xRestart THEN
				PassoChaveDuctosResfrInf01:=303;
			END_IF

		303:IF xInvDuctosInf01Habilitado THEN
				PassoChaveDuctosResfrInf01:=PassoPausaChaveDuctosResfrInf01;
			END_IF

		// Alarme Motor Parada/Reinicio
		400:xExecutaStopDuctosResfriadorInf01:=TRUE;
			PassoChaveDuctosResfrInf01:=401;

		401:xExecutaStopDuctosResfriadorInf01:=FALSE;
			xExecutaMovDuctosResfriadorInf01:=FALSE;
			PassoChaveDuctosResfrInf01:=402;

		402:IF xRestart AND xInvDuctosInf01Habilitado THEN
				PassoChaveDuctosResfrInf01:=PassoAlmChaveDuctosResfrInf01;
			END_IF

END_CASE

// BLOCOS DE EXECUÇÃO CANOPEN
//McMoveVelocityDuctosInf01(Execute:= xExecutaMovDuctosResfriadorInf01,	Velocity:=iVelocidadeDuctosResfriadorInf01,	Axis:= Resfriador_Inf01,	InVelocity=> ,	Busy=> ,CommandAborted=> , Error=> );
//McJogDuctosResfriadorInf01(Forward:= xAbreDuctosResfriadorInf01,	Backward:= xFechaDuctosResfriadorInf01, Velocity:= iVelocidadeJogDuctosResfrInf01, Axis:= Resfriador_Inf01, Done=> ,Busy=> ,CommandAborted=> ,Error=> );
//McStopDuctosResfriadorInf01(Execute:=xExecutaStopDuctosResfriadorInf01,	Axis:= Resfriador_Inf01, Done=> xStopMesaDuctosResfriadorInf01Done,Busy=> , Error=> );

ConversorPulMilimResfrInf01(
	dPulso:= 1261,
	dMilimetro:= 133,
	dEntradaPulso01:= dValorEncoderDuctosResfriadorInf01,
	iSaidaMilimetro01=> iCompAlturaAtualDuctosResfriadorInf01 );

iAlturaAtualDuctosResfriadorInf01:=iCompAlturaAtualDuctosResfriadorInf01+iCompessaAlturaDuctosResfriadorInf01;

IF xOperacaoManual THEN
	PassoHomeDuctosResfrInf01:=0;
	PassoPausaHomeDuctosResfrInf01:=0;
	PassoAlmHomeDuctosResfrInf01:=0;
	PassoAjusteDuctosResfInf01:=0;
	PassoPausaAjusteDuctosResfInf01:=0;
	PassoAlmAjusteDuctosResfInf01:=0;
	PassoChaveDuctosResfrInf01:=0;
	PassoPausaChaveDuctosResfrInf01:=0;
	PassoAlmChaveDuctosResfrInf01:=0;
	xIniciaHomeDuctosInf01:=FALSE;
	xExecutaMovDuctosResfriadorInf01:=FALSE;
	xHomeEncoderDuctosResfriadorInf01:=FALSE;
	xExecutaStopDuctosResfriadorInf01:=FALSE;
	xAbreDuctosResfriadorInf01:=FALSE;
	xFechaDuctosResfriadorInf01:=FALSE;
	xDifusorInf01Abrindo:=FALSE;
	xDifusorInf01Fechando:=FALSE;
	xAjusteAlturaDuctosInf01OK:=FALSE;
	xFechaDuctosResfriadorInf01:=FALSE;
	xBtRecAjustaAlturaDuctosInf01:=FALSE;
	BtParamDuctosResfriadorInf01:=FALSE;
	xDuctosInf01EmHome:=FALSE;
	xDuctosInf01EmAjuste:=FALSE;
	xLigaSegEstagDuctosInf01:= FALSE;
	xLigaTerEstagDuctosInf01:= FALSE;
	xReajustaAlturaDuctosInf01:=FALSE;
END_IF

(* ---- J_DuctosResfriadorInf02.prg.st ---- *)
PROGRAM J_DuctosResfriadorInf02
VAR
	PassoHomeDuctosResfrInf02: INT;
	PassoPausaHomeDuctosResfrInf02: INT;
	PassoAlmHomeDuctosResfrInf02: INT;
	PassoAjusteDuctosResfInf02: INT;
	PassoPausaAjusteDuctosResfInf02: INT;
	PassoAlmAjusteDuctosResfInf02: INT;
	PassoChaveDuctosResfrInf02: INT;
	PassoPausaChaveDuctosResfrInf02: INT;
	PassoAlmChaveDuctosResfrInf02: INT;
	///Bloco Converte Milimetro em Pulsos
	ConversorMilimPul01ResfrInf02: MmConversorPulso;
	///Bloco Converte Milimetro em Pulsos
	ConversorMilimPul02ResfrInf02: MmConversorPulso;
	///Bloco Converte Pulsos em Milimetros
	ConversorPulMilimResfrInf02: PulsoConversorMm;
	PulsoChDutosInf02Po: PulsoPositivo;
	PulsoChDutosInf02Ne: PulsoNegativo;
	xAbreDuctosResfriadorInf02: BOOL;
	xFechaDuctosResfriadorInf02: BOOL;
	xAbreResfridorInf02: BOOL;
	xFechaResfridorInf02: BOOL;
	xAjustarAlturaResfriadorInf02: BOOL;
	///Recebera uma valor fixo
	iVelocidadeHomeDuctosResfrInf02: INT;
	iVelocidadeJogDuctosResfrInf02: INT;
	iVelocidadeDuctosResfriadorInf02: INT;
	dValEncoAltura01ResfriadorInf02: DINT;
	dValEncoAltura02ResfriadorInf02: DINT;
	dValEncoAltura03ResfriadorInf02: DINT;
	dValEncoAlturaResfriadorInf02: DINT;
	dValEncoToleranciaResfrInf02: DINT;
	dValEncoAlturaVelMinimaResfrInf02: DINT := 35;
	xDifusorInf02Fechando: BOOL;
	xDifusorInf02Abrindo: BOOL;
	iCompValAltura01ResfriadorInf02: INT;
	iCompValAltura02ResfriadorInf02: INT;
	iCompValAltura03ResfriadorInf02: INT;
	iCompAlturaAtualDuctosResfriadorInf02: INT;
	iCompessaAlturaDuctosResfriadorInf02: INT;
	xPulsoChDutosInf02Po: BOOL;
	xPulsoChDutosInf02Ne: BOOL;
END_VAR

iCompessaAlturaDuctosResfriadorInf02:=REAL_TO_INT(rOffSetResfInf02);
iCompValAltura01ResfriadorInf02:=	iValAltura01ResfriadorInf02 - iCompessaAlturaDuctosResfriadorInf02;
iCompValAltura02ResfriadorInf02:=	iValAltura02ResfriadorInf02 - iCompessaAlturaDuctosResfriadorInf02;
iCompValAltura03ResfriadorInf02:=	iValAltura03ResfriadorInf02 - iCompessaAlturaDuctosResfriadorInf02;

// CONVERSÃO MILIMETROS EM PULSOS
ConversorMilimPul01ResfrInf02(
	dPulso:= 1853,
	dMilimetro:= 115,
	iEntrMilimetro01:= iCompValAltura01ResfriadorInf02,
	iEntrMilimetro02:= iCompValAltura02ResfriadorInf02,
	iEntrMilimetro03:= iCompValAltura03ResfriadorInf02,
	dSaidaPulso01=> dValEncoAltura01ResfriadorInf02,
	dSaidaPulso02=> dValEncoAltura02ResfriadorInf02,
	dSaidaPulso03=> dValEncoAltura03ResfriadorInf02);

ConversorMilimPul02ResfrInf02(
	dPulso:= 1853,
	dMilimetro:= 115,
	iEntrMilimetro01:= 2,//iValEncoToleranciaDuctosInf02,
	iEntrMilimetro02:= 10,//iValEncoAlturaVelMinimaDuctosInf02,
	dSaidaPulso01=> dValEncoToleranciaResfrInf02,
	dSaidaPulso02=> dValEncoAlturaVelMinimaResfrInf02);

// SEQUENCIA DE HOME

CASE PassoHomeDuctosResfrInf02 OF

		0:	IF xIniciaHomeDuctosInf02 OR xAutoHomeResfInf02 THEN
				PassoHomeDuctosResfrInf02:=2;
			END_IF

		2: //F xFcLimMinLimpaResfriador02 AND NOT xFcLimMaxLimpaResfriador02 THEN
				PassoHomeDuctosResfrInf02:=5;
			//ELSE
			//	PassoHomeDuctosResfrInf02:=6;
			//END_IF

		5:	IF xChAbreDuctosResfriadorInf02 THEN
				PassoHomeDuctosResfrInf02:=6;
			ELSE
				PassoHomeDuctosResfrInf02:=10;
			END_IF

		6:	xIniciaHomeDuctosInf02:=FALSE;
			xAutoHomeResfInf02:=FALSE;
			PassoHomeDuctosResfrInf02:=0;

		10:	xIniciaHomeDuctosInf02:=FALSE;
			xHomeDuctosResfriadorInf02Ok:=FALSE;
			xAjusteAlturaDuctosInf02OK:=FALSE;
			xDuctosInf02EmHome:=TRUE;
			iVelocidadeDuctosResfriadorInf02:= 150;//1*iVelocidadeHomeDuctosResfrSup02;
			PassoHomeDuctosResfrInf02:=15;

		15: xFechaResfridorInf02:=TRUE;
			PassoHomeDuctosResfrInf02:=20;

		20:	IF xSensorFechadoResfriadorInf02 THEN
				PassoHomeDuctosResfrInf02:=50;
			END_IF
			IF xPause THEN
				PassoPausaHomeDuctosResfrInf02:=10;
				PassoHomeDuctosResfrInf02:=300;
			END_IF
			IF xAlarmeMotorDifusorInf02 THEN
				PassoAlmHomeDuctosResfrInf02:=10;
				PassoHomeDuctosResfrInf02:=400;
			END_IF

		50:	xFechaResfridorInf02:=FALSE;
			PassoHomeDuctosResfrInf02:=55;

		55:	iVelocidadeDuctosResfriadorInf02:= 50;
			PassoHomeDuctosResfrInf02:=56;

		56:	xAbreResfridorInf02:=TRUE;
			PassoHomeDuctosResfrInf02:=60;

		60:	IF NOT xSensorFechadoResfriadorInf02 THEN
				PassoHomeDuctosResfrInf02:=70;
			END_IF
			IF xPause THEN
				PassoPausaHomeDuctosResfrInf02:=50;
				PassoHomeDuctosResfrInf02:=300;
			END_IF
			IF xAlarmeMotorDifusorInf02 THEN
				PassoAlmHomeDuctosResfrInf02:=50;
				PassoHomeDuctosResfrInf02:=400;
			END_IF

		70:	xAbreResfridorInf02:=FALSE;
			PassoHomeDuctosResfrInf02:=74;

		74:	IF NOT xMotorDifusorInf02Ligado THEN
				PassoHomeDuctosResfrInf02:=75;
			END_IF

		75: xHomeEncoderDuctosResfriadorInf02:=TRUE;
			PassoHomeDuctosResfrInf02:=80;

		80: xHomeEncoderDuctosResfriadorInf02:=FALSE;
			xDuctosInf02EmHome:=FALSE;
			xHomeDuctosResfriadorInf02Ok:=TRUE;
			xAutoHomeResfInf02:=FALSE;
			PassoHomeDuctosResfrInf02:=0;

		// Emergência Pausa/Reinicio
		300:xFechaResfridorInf02:=FALSE;
			xAbreResfridorInf02:=FALSE;
			PassoHomeDuctosResfrInf02:=301;

		301:xDuctosInf02EmHome:=FALSE;
			PassoHomeDuctosResfrInf02:=302;

		302:IF xRestart THEN
				PassoHomeDuctosResfrInf02:=303;
			END_IF

		303:PassoHomeDuctosResfrInf02:=0;//PassoPausaHomeDuctosResfrInf01;

		// Alarme Motor Parada/Reinicio
		400:xFechaResfridorInf02:=FALSE;
			xAbreResfridorInf02:=FALSE;
			PassoHomeDuctosResfrInf02:=401;

		401:PassoHomeDuctosResfrInf02:=402;

		402:IF xRestart AND iCanOpenInverDuctResfrInf02StateOk THEN
				PassoHomeDuctosResfrInf02:=PassoAlmHomeDuctosResfrInf02;
			END_IF
END_CASE

//
IF xTerceiroEstagioResfriador THEN
	dValEncoAlturaResfriadorInf02:=dValEncoAltura03ResfriadorInf02;
ELSIF xSegundoEstagioResfriador THEN
	dValEncoAlturaResfriadorInf02:=dValEncoAltura02ResfriadorInf02;
ELSE
	dValEncoAlturaResfriadorInf02:=dValEncoAltura01ResfriadorInf02;
END_IF

// SEQUENCIA DE FUNCIONAMENTO

IF (xBtRecAjustaAlturaDuctosInf02 OR BtParamDuctosResfriadorInf02 OR (xLigaSegEstagDuctosInf02 AND NOT xChAbreDuctosResfriadorInf02) OR (xLigaTerEstagDuctosInf02 AND NOT xChAbreDuctosResfriadorInf02) OR xReajustaAlturaDuctosInf02) AND xHomeDuctosResfriadorInf02Ok THEN
	xAjustarAlturaResfriadorInf02:=TRUE;
	xBtRecAjustaAlturaDuctosInf02:=FALSE;
	BtParamDuctosResfriadorInf02:=FALSE;
	xLigaSegEstagDuctosInf02:= FALSE;
	xLigaTerEstagDuctosInf02:= FALSE;
	xReajustaAlturaDuctosInf02:=FALSE;
ELSE
	xBtRecAjustaAlturaDuctosInf02:=FALSE;
	BtParamDuctosResfriadorInf02:=FALSE;
	xLigaSegEstagDuctosInf02:= FALSE;
	xLigaTerEstagDuctosInf02:= FALSE;
	xReajustaAlturaDuctosInf02:=FALSE;
END_IF

CASE PassoAjusteDuctosResfInf02 OF

		0:	IF xAjustarAlturaResfriadorInf02 AND NOT xAbreDuctosResfriadorInf02 THEN //AND NOT xChAbreDuctosResfriadorInf02 THEN
				PassoAjusteDuctosResfInf02:=10;
			END_IF

		10:	xAjustarAlturaResfriadorInf02:=FALSE;
			xAjusteAlturaDuctosInf02OK:=FALSE;
			xDuctosInf02EmAjuste:=TRUE;
			IF dValorEncoderDuctosResfriadorInf02<dValEncoAlturaResfriadorInf02-dValEncoToleranciaResfrInf02 THEN
				xDifusorInf02Abrindo:=TRUE;
				PassoAjusteDuctosResfInf02:=20;//Abre
			END_IF
			IF dValorEncoderDuctosResfriadorInf02>dValEncoAlturaResfriadorInf02+dValEncoToleranciaResfrInf02 THEN
				PassoAjusteDuctosResfInf02:=100;//Fecha
				xDifusorInf02Fechando:=TRUE;
			END_IF
			IF dValorEncoderDuctosResfriadorInf02>=dValEncoAlturaResfriadorInf02-dValEncoToleranciaResfrInf02 AND dValorEncoderDuctosResfriadorInf02<=dValEncoAlturaResfriadorInf02+dValEncoToleranciaResfrInf02 THEN
				PassoAjusteDuctosResfInf02:=180;//Não se Move
			END_IF
//Abre
		20:	iVelocidadeDuctosResfriadorInf02:= iVelocidadeAjusteDuctosResfriadorInf02;
			PassoAjusteDuctosResfInf02:=25;

		25:	xAbreResfridorInf02:=TRUE;
			PassoAjusteDuctosResfInf02:=30;

		30:	IF (dValorEncoderDuctosResfriadorInf02>=dValEncoAlturaResfriadorInf02-35(*dValEncoAlturaVelMinimaResfrInf02*)) OR xSensorAbertoResfriadorInf02 THEN
				PassoAjusteDuctosResfInf02:=40;
			END_IF
			IF iVelocidadeDuctosResfriadorInf02<> iVelocidadeAjusteDuctosResfriadorInf02 THEN
				PassoAjusteDuctosResfInf02:=20;
			END_IF
			IF xPause THEN
				PassoPausaAjusteDuctosResfInf02:=20;
				PassoAjusteDuctosResfInf02:=300;
			END_IF
			IF xAlarmeMotorDifusorInf02 THEN
				PassoAlmAjusteDuctosResfInf02:=20;
				PassoAjusteDuctosResfInf02:=400;
			END_IF

		40:	iVelocidadeDuctosResfriadorInf02:= iVelocidadeMinimaDuctosResfriadorInf02;
			PassoAjusteDuctosResfInf02:=50;

		50:	IF (dValorEncoderDuctosResfriadorInf02>=dValEncoAlturaResfriadorInf02) OR xSensorAbertoResfriadorInf02 THEN
				PassoAjusteDuctosResfInf02:=60;
			END_IF
			IF xPause THEN
				PassoPausaAjusteDuctosResfInf02:=40;
				PassoAjusteDuctosResfInf02:=300;
			END_IF
			IF xAlarmeMotorDifusorInf02 THEN
				PassoAlmAjusteDuctosResfInf02:=40;
				PassoAjusteDuctosResfInf02:=400;
			END_IF

		60: xAbreResfridorInf02:=FALSE;
			PassoAjusteDuctosResfInf02:=180;

//Desce
		100:iVelocidadeDuctosResfriadorInf02:= 1*iVelocidadeAjusteDuctosResfriadorInf02;
			PassoAjusteDuctosResfInf02:=105;

		105:xFechaResfridorInf02:=TRUE;
			PassoAjusteDuctosResfInf02:=110;

		110:IF (dValorEncoderDuctosResfriadorInf02 <= dValEncoAlturaResfriadorInf02+35(*dValEncoAlturaVelMinimaResfrInf02*)) OR xSensorFechadoResfriadorInf02 THEN
				PassoAjusteDuctosResfInf02:=120;
			END_IF
			IF iVelocidadeDuctosResfriadorInf02<> 1*iVelocidadeAjusteDuctosResfriadorInf02 THEN
				PassoAjusteDuctosResfInf02:=100;
			END_IF
			IF xPause THEN
				PassoPausaAjusteDuctosResfInf02:=100;
				PassoAjusteDuctosResfInf02:=300;
			END_IF
			IF xAlarmeMotorDifusorInf02 THEN
				PassoAlmAjusteDuctosResfInf02:=100;
				PassoAjusteDuctosResfInf02:=400;
			END_IF

		120:iVelocidadeDuctosResfriadorInf02:= 1*iVelocidadeMinimaDuctosResfriadorInf02;
			PassoAjusteDuctosResfInf02:=130;

		130:IF (dValorEncoderDuctosResfriadorInf02<=dValEncoAlturaResfriadorInf02) OR xSensorFechadoResfriadorInf02 THEN
				PassoAjusteDuctosResfInf02:=140;
			END_IF
			IF iVelocidadeDuctosResfriadorInf02<> 1*iVelocidadeMinimaDuctosResfriadorInf02 THEN
				PassoAjusteDuctosResfInf02:=120;
			END_IF
			IF xPause THEN
				PassoPausaAjusteDuctosResfInf02:=120;
				PassoAjusteDuctosResfInf02:=300;
			END_IF
			IF xAlarmeMotorDifusorInf02 THEN
				PassoAlmAjusteDuctosResfInf02:=120;
				PassoAjusteDuctosResfInf02:=400;
			END_IF

		140:xFechaResfridorInf02:=FALSE;
			PassoAjusteDuctosResfInf02:=180;
//Fim
		180:xDifusorInf02Abrindo:=FALSE;
			xDifusorInf02Fechando:=FALSE;
			xDuctosInf02EmAjuste:=FALSE;
			xAjusteAlturaDuctosInf02OK:=TRUE;
			PassoAjusteDuctosResfInf02:=0;

		// Emergência Pausa/Reinicio
		300:xAbreResfridorInf02:=FALSE;
			xFechaResfridorInf02:=FALSE;
			PassoAjusteDuctosResfInf02:=301;

		301:PassoAjusteDuctosResfInf02:=302;

		302:IF xRestart THEN
				PassoAjusteDuctosResfInf02:=303;
			END_IF

		303:PassoAjusteDuctosResfInf02:=PassoPausaAjusteDuctosResfInf02;

		// Alarme Motor Parada/Reinicio
		400:xAbreResfridorInf02:=FALSE;
			xFechaResfridorInf02:=FALSE;
			PassoAjusteDuctosResfInf02:=401;

		401:PassoAjusteDuctosResfInf02:=402;

		402:IF xRestart AND iCanOpenInverDuctResfrInf02StateOk THEN
				PassoAjusteDuctosResfInf02:=PassoAlmAjusteDuctosResfInf02;
			END_IF

END_CASE

// MOVIMENTO COM A CHAVE DE ABERTURA

PulsoChDutosInf02Po(Entrada:= xChAbreDuctosResfriadorInf02, SaidaPulsoPo=> xPulsoChDutosInf02Po);
PulsoChDutosInf02Ne(Entrada:= xChAbreDuctosResfriadorInf02, SaidaPulsoNe=> xPulsoChDutosInf02Ne);

(*IF xPulsoChDutosInf02Po THEN
	xPausaMesaResfrimento:=TRUE;
END_IF
IF xPulsoChDutosInf02Ne THEN
	xPausaMesaResfrimento:=FALSE;
END_IF*)

CASE PassoChaveDuctosResfrInf02 OF

		0:	IF xPulsoChDutosInf02Po AND xHomeDuctosResfriadorInf02Ok THEN //IF xChAbreDuctosResfriadorInf02 AND xHomeDuctosResfriadorInf02Ok THEN
				PassoChaveDuctosResfrInf02:=5;
				PassoAjusteDuctosResfInf02:=0;
				xFechaResfridorInf02:=FALSE;
			END_IF

		5:	IF NOT xPrimeiroEstagioResfriador THEN
				PassoChaveDuctosResfrInf02:=10;
			END_IF

		10:	iVelocidadeJogDuctosResfrInf02:=iVelocidadeAjusteDuctosResfriadorInf02;
			xAjusteAlturaDuctosInf02OK:=FALSE;
			xAbreDuctosResfriadorInf02:=TRUE;
			IF xSensorAbertoResfriadorInf02 THEN
				PassoChaveDuctosResfrInf02:=20;
			END_IF
			IF xPause THEN
				PassoPausaChaveDuctosResfrInf02:=10;
				PassoChaveDuctosResfrInf02:=300;
			END_IF
			IF xAlarmeMotorDifusorInf02 THEN
				PassoAlmChaveDuctosResfrInf02:=10;
				PassoChaveDuctosResfrInf02:=400;
			END_IF

		20:	xAbreDuctosResfriadorInf02:=FALSE;
			PassoChaveDuctosResfrInf02:=21;

		21:	IF xPulsoChDutosInf02Ne THEN//IF NOT xChAbreDuctosResfriadorInf02 THEN
				xAbreDuctosResfriadorInf02:=FALSE;
				PassoChaveDuctosResfrInf02:=0;
				PassoAjusteDuctosResfInf02:=100;
			END_IF
			IF xPause THEN
				PassoPausaChaveDuctosResfrInf02:=21;
				PassoChaveDuctosResfrInf02:=300;
			END_IF
			IF xAlarmeMotorDifusorInf02 THEN
				PassoAlmChaveDuctosResfrInf02:=21;
				PassoChaveDuctosResfrInf02:=400;
			END_IF

		// Emergência Pausa/Reinicio
		300:xAbreDuctosResfriadorInf02:=FALSE;
			PassoChaveDuctosResfrInf02:=301;

		301:PassoChaveDuctosResfrInf02:=302;

		302:IF xRestart THEN
				PassoChaveDuctosResfrInf02:=303;
			END_IF

		303:PassoChaveDuctosResfrInf02:=PassoPausaChaveDuctosResfrInf02;

		// Alarme Motor Parada/Reinicio
		400:xAbreDuctosResfriadorInf02:=FALSE;
			PassoChaveDuctosResfrInf02:=401;

		401:PassoChaveDuctosResfrInf02:=402;

		402:IF xRestart AND iCanOpenInverDuctResfrInf02StateOk THEN
				PassoChaveDuctosResfrInf02:=PassoAlmChaveDuctosResfrInf02;
			END_IF

END_CASE

// MOVIMENTAÇÃO PELO COMANDO ENTRADAS DIGITAIS DO INVERSOR
// Comando e Dirreção
xMotorResfridorInf02Abre:= xAbreResfridorInf02 OR xAbreDuctosResfriadorInf02;
xMotorResfridorInf02Fecha:= xFechaResfridorInf02;

InversorResfInf02.i_xAvanco:=xMotorResfridorInf02Abre;
InversorResfInf02.i_xRecuo:=xMotorResfridorInf02Fecha;
// Velocidade
InversorResfInf02.i_iFreqRef:=iVelocidadeDuctosResfriadorInf02;
//---------------------------------------------------------------------------------\\

ConversorPulMilimResfrInf02(
	dPulso:= 1853,
	dMilimetro:= 115,
	dEntradaPulso01:= dValorEncoderDuctosResfriadorInf02,
	iSaidaMilimetro01=> iCompAlturaAtualDuctosResfriadorInf02 );

iAlturaAtualDuctosResfriadorInf02:=iCompAlturaAtualDuctosResfriadorInf02+iCompessaAlturaDuctosResfriadorInf02;

IF xOperacaoManual THEN
	PassoHomeDuctosResfrInf02:=0;
	PassoPausaHomeDuctosResfrInf02:=0;
	PassoAlmHomeDuctosResfrInf02:=0;
	PassoAjusteDuctosResfInf02:=0;
	PassoPausaAjusteDuctosResfInf02:=0;
	PassoAlmAjusteDuctosResfInf02:=0;
	PassoChaveDuctosResfrInf02:=0;
	PassoPausaChaveDuctosResfrInf02:=0;
	PassoAlmChaveDuctosResfrInf02:=0;
	xIniciaHomeDuctosInf02:=FALSE;
	xHomeEncoderDuctosResfriadorInf02:=FALSE;
	xAbreDuctosResfriadorInf02:=FALSE;
	xFechaDuctosResfriadorInf02:=FALSE;
	xDifusorInf02Abrindo:=FALSE;
	xDifusorInf02Fechando:=FALSE;
	xAjusteAlturaDuctosInf02OK:=FALSE;
	xFechaDuctosResfriadorInf02:=FALSE;
	xBtRecAjustaAlturaDuctosInf02:=FALSE;
	BtParamDuctosResfriadorInf02:=FALSE;
	xDuctosInf02EmHome:=FALSE;
	xDuctosInf02EmAjuste:=FALSE;
	xLigaSegEstagDuctosInf02:= FALSE;
	xLigaTerEstagDuctosInf02:= FALSE;
	xReajustaAlturaDuctosInf02:=FALSE;

	xFechaResfridorInf02:=FALSE;
	xAbreResfridorInf02:=FALSE;
	xLigaTerEstagDuctosInf02:=FALSE;
END_IF

(* ---- J_DuctosResfriadorSup01.prg.st ---- *)
PROGRAM J_DuctosResfriadorSup01
VAR
	PassoHomeDuctosResfrSup01: INT;
	PassoPausaHomeDuctosResfrSup01: INT;
	PassoAlmHomeDuctosResfrSup01: INT;
	PassoAjusteDuctosResfSup01: INT;
	PassoPausaAjusteDuctosResfSup01: INT;
	PassoAlmAjusteDuctosResfSup01: INT;
	PassoChaveDuctosResfrSup01: INT;
	PassoPausaChaveDuctosResfrSup01: INT;
	PassoAlmChaveDuctosResfrSup01: INT;
	///Bloco Converte Milimetro em Pulsos
	ConversorMilimPul01ResfrSup01: MmConversorPulso;
	///Bloco Converte Milimetro em Pulsos
	ConversorMilimPul02ResfrSup01: MmConversorPulso;
	///Bloco Converte Pulsos em Milimetros
	ConversorPulMilimResfrSup01: PulsoConversorMm;
	PulsoChDutosSup01Po: PulsoPositivo;
	PulsoChDutosSup01Ne: PulsoNegativo;
	xAbreDuctosResfriadorSup01: BOOL;
	xFechaDuctosResfriadorSup01: BOOL;
	xAbreResfridorSup01: BOOL;
	xFechaResfridorSup01: BOOL;
	xAjustarAlturaResfriadorSup01: BOOL;
	///Recebera uma valor fixo
	iVelocidadeHomeDuctosResfrSup01: INT;
	iVelocidadeJogDuctosResfrSup01: INT;
	iVelocidadeDuctosResfriadorSup01: INT;
	dValEncoAltura01ResfriadorSup01: DINT;
	dValEncoAltura02ResfriadorSup01: DINT;
	dValEncoAltura03ResfriadorSup01: DINT;
	dValEncoAlturaResfriadorSup01: DINT;
	dValEncoToleranciaResfrSup01: DINT;
	dValEncoAlturaVelMinimaResfrSup01: DINT := 35;
	xDifusorSup01Fechando: BOOL;
	xDifusorSup01Abrindo: BOOL;
	iCompValAltura01ResfriadorSup01: INT;
	iCompValAltura02ResfriadorSup01: INT;
	iCompValAltura03ResfriadorSup01: INT;
	iCompAlturaAtualDuctosResfriadorSup01: INT;
	iCompessaAlturaDuctosResfriadorSup01: INT;
	xPulsoChDutosSup01Po: BOOL;
	xPulsoChDutosSup01Ne: BOOL;
END_VAR

iCompessaAlturaDuctosResfriadorSup01:=REAL_TO_INT(rOffSetResfSup01);
iCompValAltura01ResfriadorSup01:=	iValAltura01ResfriadorSup01 - iCompessaAlturaDuctosResfriadorSup01;
iCompValAltura02ResfriadorSup01:=	iValAltura02ResfriadorSup01 - iCompessaAlturaDuctosResfriadorSup01;
iCompValAltura03ResfriadorSup01:=	iValAltura03ResfriadorSup01 - iCompessaAlturaDuctosResfriadorSup01;

// CONVERSÃO MILIMETROS EM PULSOS
ConversorMilimPul01ResfrSup01(
	dPulso:= 257614,
	dMilimetro:= 33,
	iEntrMilimetro01:= iCompValAltura01ResfriadorSup01,
	iEntrMilimetro02:= iCompValAltura02ResfriadorSup01,
	iEntrMilimetro03:= iCompValAltura03ResfriadorSup01,
	dSaidaPulso01=> dValEncoAltura01ResfriadorSup01,
	dSaidaPulso02=> dValEncoAltura02ResfriadorSup01,
	dSaidaPulso03=> dValEncoAltura03ResfriadorSup01);

ConversorMilimPul02ResfrSup01(
	dPulso:= 257614,
	dMilimetro:= 33,
	iEntrMilimetro01:= 2,//iValEncoToleranciaDuctosSup01,
	iEntrMilimetro02:= 8,//iValEncoAlturaVelMinimaDuctosSup01,
	dSaidaPulso01=> dValEncoToleranciaResfrSup01,
	dSaidaPulso02=> dValEncoAlturaVelMinimaResfrSup01);

// SEQUENCIA DE HOME

CASE PassoHomeDuctosResfrSup01 OF

		0:	IF xIniciaHomeDuctosSup01 THEN
				PassoHomeDuctosResfrSup01:=10;//5;
			END_IF

		5:	IF xChAbreDuctosResfriadorSup01 THEN
				PassoHomeDuctosResfrSup01:=6;
			ELSE
				PassoHomeDuctosResfrSup01:=10;
			END_IF

		6:	xIniciaHomeDuctosSup01:=FALSE;
			PassoHomeDuctosResfrSup01:=0;

		10:	xIniciaHomeDuctosSup01:=FALSE;
			xHomeDuctosResfriadorSup01Ok:=FALSE;
			xAjusteAlturaDuctosSup01OK:=FALSE;
			xDuctosSup01EmHome:=TRUE;
			iVelocidadeDuctosResfriadorSup01:= 150;//1*iVelocidadeHomeDuctosResfr;
			PassoHomeDuctosResfrSup01:=15;

		15: xFechaResfridorSup01:=TRUE;
			PassoHomeDuctosResfrSup01:=20;

		20:	IF xSensorFechadoResfriadorSup01 THEN
				PassoHomeDuctosResfrSup01:=50;
			END_IF
			IF xPause THEN
				PassoPausaHomeDuctosResfrSup01:=10;
				PassoHomeDuctosResfrSup01:=300;
			END_IF
			IF xAlarmeMotorDifusorSup01 THEN
				PassoAlmHomeDuctosResfrSup01:=10;
				PassoHomeDuctosResfrSup01:=400;
			END_IF

		50:	xFechaResfridorSup01:=FALSE;
			PassoHomeDuctosResfrSup01:=55;

		55:	iVelocidadeDuctosResfriadorSup01:= 50;
			PassoHomeDuctosResfrSup01:=56;

		56:	xAbreResfridorSup01:=TRUE;
			PassoHomeDuctosResfrSup01:=60;

		60:	IF NOT xSensorFechadoResfriadorSup01 THEN
				PassoHomeDuctosResfrSup01:=70;
			END_IF
			IF xPause THEN
				PassoPausaHomeDuctosResfrSup01:=50;
				PassoHomeDuctosResfrSup01:=300;
			END_IF
			IF xAlarmeMotorDifusorSup01 THEN
				PassoAlmHomeDuctosResfrSup01:=50;
				PassoHomeDuctosResfrSup01:=400;
			END_IF

		70:	xAbreResfridorSup01:=FALSE;
			PassoHomeDuctosResfrSup01:=74;

		74:	IF NOT xMotorDifusorSup01Ligado THEN
				PassoHomeDuctosResfrSup01:=75;
			END_IF

		75: xHomeEncoderDuctosResfriadorSup01:=TRUE;
			PassoHomeDuctosResfrSup01:=80;

		80: xHomeEncoderDuctosResfriadorSup01:=FALSE;
			xDuctosSup01EmHome:=FALSE;
			xHomeDuctosResfriadorSup01Ok:=TRUE;

		// Emergência Pausa/Reinicio
		300:xFechaResfridorSup01:=FALSE;
			xAbreResfridorSup01:=FALSE;
			PassoHomeDuctosResfrSup01:=301;

		301:xDuctosSup01EmHome:=FALSE;
			PassoHomeDuctosResfrSup01:=302;

		302:IF xRestart THEN
				PassoHomeDuctosResfrSup01:=303;
			END_IF

		303:PassoHomeDuctosResfrSup01:=0;//PassoPausaHomeDuctosResfr;

		// Alarme Motor Parada/Reinicio
		400:xFechaResfridorSup01:=FALSE;
			xAbreResfridorSup01:=FALSE;
			PassoHomeDuctosResfrSup01:=401;

		401:PassoHomeDuctosResfrSup01:=402;

		402:IF xRestart AND iCanOpenInverDuctResfrSup01StateOk THEN
				PassoHomeDuctosResfrSup01:=PassoAlmHomeDuctosResfrSup01;
			END_IF
END_CASE

//IF xTerceiroEstagioResfriador THEN
//	dValEncoAlturaResfriadorSup01:=dValEncoAltura03ResfriadorSup01;
//ELSIF xSegundoEstagioResfriador THEN
//	dValEncoAlturaResfriadorSup01:=dValEncoAltura02ResfriadorSup01;
//ELSE
	dValEncoAlturaResfriadorSup01:=dValEncoAltura01ResfriadorSup01;
//END_IF

// SEQUENCIA DE FUNCIONAMENTO

IF (xBtRecAjustaAlturaDuctosSup01 OR BtParamDuctosResfriadorSup01 OR xLigaSegEstagDuctosSup01 OR xLigaTerEstagDuctosSup01 OR xReajustaAlturaDuctosSup01) AND xHomeDuctosResfriadorSup01Ok THEN
	xAjustarAlturaResfriadorSup01:=TRUE;
	xBtRecAjustaAlturaDuctosSup01:=FALSE;
	BtParamDuctosResfriadorSup01:=FALSE;
	xLigaSegEstagDuctosSup01:= FALSE;
	xLigaTerEstagDuctosSup01:= FALSE;
	xReajustaAlturaDuctosSup01:=FALSE;
ELSE
	xBtRecAjustaAlturaDuctosSup01:=FALSE;
	BtParamDuctosResfriadorSup01:=FALSE;
	xLigaSegEstagDuctosSup01:= FALSE;
	xLigaTerEstagDuctosSup01:= FALSE;
	xReajustaAlturaDuctosSup01:=FALSE;
END_IF

CASE PassoAjusteDuctosResfSup01 OF

		0:	IF xAjustarAlturaResfriadorSup01 (*AND NOT xChAbreDuctosResfriadorSup01*) THEN
				PassoAjusteDuctosResfSup01:=10;
			END_IF

		10:	xAjustarAlturaResfriadorSup01:=FALSE;
			xAjusteAlturaDuctosSup01OK:=FALSE;
			xDuctosSup01EmAjuste:=TRUE;
			IF dValorEncoderDuctosResfriadorSup01<dValEncoAlturaResfriadorSup01-dValEncoToleranciaResfrSup01 THEN
				xDifusorSup01Abrindo:=TRUE;
				PassoAjusteDuctosResfSup01:=20;//Sobe
			END_IF
			IF dValorEncoderDuctosResfriadorSup01>dValEncoAlturaResfriadorSup01+dValEncoToleranciaResfrSup01 THEN
				PassoAjusteDuctosResfSup01:=100;//Desce
				xDifusorSup01Fechando:=TRUE;
			END_IF
			IF dValorEncoderDuctosResfriadorSup01>=dValEncoAlturaResfriadorSup01-dValEncoToleranciaResfrSup01 AND dValorEncoderDuctosResfriadorSup01<=dValEncoAlturaResfriadorSup01+dValEncoToleranciaResfrSup01 THEN
				PassoAjusteDuctosResfSup01:=180;//Não se Move
			END_IF
//Sobe
		20:	iVelocidadeDuctosResfriadorSup01:= iVelocidadeAjusteDuctosResfriadorSup01;
			PassoAjusteDuctosResfSup01:=25;

		25:	xAbreResfridorSup01:=TRUE;
			PassoAjusteDuctosResfSup01:=30;

		30:	IF (dValorEncoderDuctosResfriadorSup01>=dValEncoAlturaResfriadorSup01-35(*dValEncoAlturaVelMinimaResfrSup01*)) OR xSensorAbertoResfriadorSup01 THEN
				PassoAjusteDuctosResfSup01:=40;
			END_IF
			IF iVelocidadeDuctosResfriadorSup01<> iVelocidadeAjusteDuctosResfriadorSup01 THEN
				PassoAjusteDuctosResfSup01:=20;
			END_IF
			IF xPause THEN
				PassoPausaAjusteDuctosResfSup01:=20;
				PassoAjusteDuctosResfSup01:=300;
			END_IF
			IF xAlarmeMotorDifusorSup01 THEN
				PassoAlmAjusteDuctosResfSup01:=20;
				PassoAjusteDuctosResfSup01:=400;
			END_IF

		40:	iVelocidadeDuctosResfriadorSup01:= iVelocidadeMinimaDuctosResfriadorSup01;
			PassoAjusteDuctosResfSup01:=50;

		50:	IF (dValorEncoderDuctosResfriadorSup01>=dValEncoAlturaResfriadorSup01) OR xSensorAbertoResfriadorSup01 THEN
				PassoAjusteDuctosResfSup01:=60;
			END_IF
			IF xPause THEN
				PassoPausaAjusteDuctosResfSup01:=40;
				PassoAjusteDuctosResfSup01:=300;
			END_IF
			IF xAlarmeMotorDifusorSup01 THEN
				PassoAlmAjusteDuctosResfSup01:=40;
				PassoAjusteDuctosResfSup01:=400;
			END_IF

		60: xAbreResfridorSup01:=FALSE;
			PassoAjusteDuctosResfSup01:=180;

//Desce
		100:iVelocidadeDuctosResfriadorSup01:= 1*iVelocidadeAjusteDuctosResfriadorSup01;
			PassoAjusteDuctosResfSup01:=105;

		105:xFechaResfridorSup01:=TRUE;
			PassoAjusteDuctosResfSup01:=110;

		110:IF (dValorEncoderDuctosResfriadorSup01 <= dValEncoAlturaResfriadorSup01+35(*dValEncoAlturaVelMinimaResfrSup01*)) OR xSensorFechadoResfriadorSup01 THEN
				PassoAjusteDuctosResfSup01:=120;
			END_IF
			IF iVelocidadeDuctosResfriadorSup01<> 1*iVelocidadeAjusteDuctosResfriadorSup01 THEN
				PassoAjusteDuctosResfSup01:=100;
			END_IF
			IF xPause THEN
				PassoPausaAjusteDuctosResfSup01:=100;
				PassoAjusteDuctosResfSup01:=300;
			END_IF
			IF xAlarmeMotorDifusorSup01 THEN
				PassoAlmAjusteDuctosResfSup01:=100;
				PassoAjusteDuctosResfSup01:=400;
			END_IF

		120:iVelocidadeDuctosResfriadorSup01:= 1*iVelocidadeMinimaDuctosResfriadorSup01;
			PassoAjusteDuctosResfSup01:=130;

		130:IF (dValorEncoderDuctosResfriadorSup01<=dValEncoAlturaResfriadorSup01) OR xSensorFechadoResfriadorSup01 THEN
				PassoAjusteDuctosResfSup01:=140;
			END_IF
			IF iVelocidadeDuctosResfriadorSup01<> 1*iVelocidadeMinimaDuctosResfriadorSup01 THEN
				PassoAjusteDuctosResfSup01:=120;
			END_IF
			IF xPause THEN
				PassoPausaAjusteDuctosResfSup01:=120;
				PassoAjusteDuctosResfSup01:=300;
			END_IF
			IF xAlarmeMotorDifusorSup01 THEN
				PassoAlmAjusteDuctosResfSup01:=120;
				PassoAjusteDuctosResfSup01:=400;
			END_IF

		140:xFechaResfridorSup01:=FALSE;
			PassoAjusteDuctosResfSup01:=180;
//Fim
		180:xDifusorSup01Abrindo:=FALSE;
			xDifusorSup01Fechando:=FALSE;
			xDuctosSup01EmAjuste:=FALSE;
			xAjusteAlturaDuctosSup01OK:=TRUE;
			PassoAjusteDuctosResfSup01:=0;

		// Emergência Pausa/Reinicio
		300:xAbreResfridorSup01:=FALSE;
			xFechaResfridorSup01:=FALSE;
			PassoAjusteDuctosResfSup01:=301;

		301:PassoAjusteDuctosResfSup01:=302;

		302:IF xRestart THEN
				PassoAjusteDuctosResfSup01:=303;
			END_IF

		303:PassoAjusteDuctosResfSup01:=PassoPausaAjusteDuctosResfSup01;

		// Alarme Motor Parada/Reinicio
		400:xAbreResfridorSup01:=FALSE;
			xFechaResfridorSup01:=FALSE;
			PassoAjusteDuctosResfSup01:=401;

		401:PassoAjusteDuctosResfSup01:=402;

		402:IF xRestart AND iCanOpenInverDuctResfrSup01StateOk THEN
				PassoAjusteDuctosResfSup01:=PassoAlmAjusteDuctosResfSup01;
			END_IF

END_CASE

// MOVIMENTO COM A CHAVE DE ABERTURA

(*PulsoChDutosSup01Po(Entrada:= xChAbreDuctosResfriadorSup01, SaidaPulsoPo=> xPulsoChDutosSup01Po);
PulsoChDutosSup01Ne(Entrada:= xChAbreDuctosResfriadorSup01, SaidaPulsoNe=> xPulsoChDutosSup01Ne);

IF xPulsoChDutosSup01Po THEN
	xPausaMesaResfrimento:=TRUE;
END_IF
IF xPulsoChDutosSup01Ne THEN
	xPausaMesaResfrimento:=FALSE;
END_IF

CASE PassoChaveDuctosResfrSup01 OF

		0:	IF xChAbreDuctosResfriadorSup01 AND xHomeDuctosResfriadorSup01Ok THEN
				PassoChaveDuctosResfrSup01:=10;
				PassoAjusteDuctosResfSup01:=0;
				xFechaResfridorSup01:=FALSE;
				END_IF

		5:	IF NOT xPrimeiroEstagioResfriador THEN
				PassoChaveDuctosResfrSup01:=10;
			END_IF

		10:	iVelocidadeJogDuctosResfrSup01:=iVelocidadeAjusteDuctosResfriadorSup01;
			xAjusteAlturaDuctosSup01OK:=FALSE;
			xAbreDuctosResfriadorSup01:=TRUE;
			IF xSensorAbertoResfriadorSup01 THEN
				PassoChaveDuctosResfrSup01:=20;
			END_IF
			IF xPause THEN
				PassoPausaChaveDuctosResfrSup01:=10;
				PassoChaveDuctosResfrSup01:=300;
			END_IF
			IF xAlarmeMotorDifusorSup01 THEN
				PassoAlmChaveDuctosResfrSup01:=10;
				PassoChaveDuctosResfrSup01:=400;
			END_IF

		20:	xAbreDuctosResfriadorSup01:=FALSE;
			PassoChaveDuctosResfrSup01:=21;

		21:	IF xPulsoChDutosSup01Ne THEN//IF NOT xChAbreDuctosResfriadorSup02 THEN
				xAbreDuctosResfriadorSup01:=FALSE;
				PassoChaveDuctosResfrSup01:=0;
				PassoAjusteDuctosResfSup01:=100;
			END_IF
			IF xPause THEN
				PassoPausaChaveDuctosResfrSup01:=21;
				PassoChaveDuctosResfrSup01:=300;
			END_IF
			IF xAlarmeMotorDifusorSup01 THEN
				PassoAlmChaveDuctosResfrSup01:=21;
				PassoChaveDuctosResfrSup01:=400;
			END_IF

		// Emergência Pausa/Reinicio
		300:xAbreDuctosResfriadorSup01:=FALSE;
			PassoChaveDuctosResfrSup01:=301;

		301:PassoChaveDuctosResfrSup01:=302;

		302:IF xRestart THEN
				PassoChaveDuctosResfrSup01:=303;
			END_IF

		303:PassoChaveDuctosResfrSup01:=PassoPausaChaveDuctosResfrSup01;

		// Alarme Motor Parada/Reinicio
		400:xAbreDuctosResfriadorSup01:=FALSE;
			PassoChaveDuctosResfrSup01:=401;

		401:PassoChaveDuctosResfrSup01:=402;

		402:IF xRestart AND iCanOpenInverDuctResfrSup01StateOk THEN
				PassoChaveDuctosResfrSup01:=PassoAlmChaveDuctosResfrSup01;
			END_IF

END_CASE
*)
// MOVIMENTAÇÃO PELO COMANDO ENTRADAS DIGITAIS DO INVERSOR
// Comando e Direção
xMotorResfridorSup01Abre:= xAbreResfridorSup01 OR xAbreDuctosResfriadorSup01;
xMotorResfridorSup01Fecha:= xFechaResfridorSup01;

InversorResfSup01.i_xAvanco:=xMotorResfridorSup01Abre;
InversorResfSup01.i_xRecuo:=xMotorResfridorSup01Fecha;
// Velocidade
InversorResfSup01.i_iFreqRef:=iVelocidadeDuctosResfriadorSup01;
//---------------------------------------------------------------------------------\\

ConversorPulMilimResfrSup01(
	dPulso:= 257614,
	dMilimetro:= 33,
	dEntradaPulso01:= dValorEncoderDuctosResfriadorSup01,
	iSaidaMilimetro01=> iCompAlturaAtualDuctosResfriadorSup01 );

iAlturaAtualDuctosResfriadorSup01:=iCompAlturaAtualDuctosResfriadorSup01+iCompessaAlturaDuctosResfriadorSup01;

IF xOperacaoManual THEN
	PassoHomeDuctosResfrSup01:=0;
	PassoPausaHomeDuctosResfrSup01:=0;
	PassoAlmHomeDuctosResfrSup01:=0;
	PassoAjusteDuctosResfSup01:=0;
	PassoPausaAjusteDuctosResfSup01:=0;
	PassoAlmAjusteDuctosResfSup01:=0;
	PassoChaveDuctosResfrSup01:=0;
	PassoPausaChaveDuctosResfrSup01:=0;
	PassoAlmChaveDuctosResfrSup01:=0;
	xIniciaHomeDuctosSup01:=FALSE;
	xHomeEncoderDuctosResfriadorSup01:=FALSE;
	xAbreDuctosResfriadorSup01:=FALSE;
	xFechaDuctosResfriadorSup01:=FALSE;
	xDifusorSup01Abrindo:=FALSE;
	xDifusorSup01Fechando:=FALSE;
	xAjusteAlturaDuctosSup01OK:=FALSE;
	xFechaDuctosResfriadorSup01:=FALSE;
	xBtRecAjustaAlturaDuctosSup01:=FALSE;
	BtParamDuctosResfriadorSup01:=FALSE;
	xDuctosSup01EmHome:=FALSE;
	xDuctosSup01EmAjuste:=FALSE;
	xLigaSegEstagDuctosSup01:= FALSE;
	xLigaTerEstagDuctosSup01:= FALSE;
	xReajustaAlturaDuctosSup01:=FALSE;
	xFechaResfridorSup01:=FALSE;
	xAbreResfridorSup01:=FALSE;
	xFechaResfridorSup01:=FALSE;
	xAbreResfridorSup01:=FALSE;
	xLigaTerEstagDuctosSup01:=FALSE;
END_IF

(* ---- J_DuctosResfriadorSup02.prg.st ---- *)
PROGRAM J_DuctosResfriadorSup02
VAR
	PassoHomeDuctosResfrSup02: INT;
	PassoPausaHomeDuctosResfrSup02: INT;
	PassoAlmHomeDuctosResfrSup02: INT;
	PassoAjusteDuctosResfSup02: INT;
	PassoPausaAjusteDuctosResfSup02: INT;
	PassoAlmAjusteDuctosResfSup02: INT;
	PassoChaveDuctosResfrSup02: INT;
	PassoPausaChaveDuctosResfrSup02: INT;
	PassoAlmChaveDuctosResfrSup02: INT;
	///Bloco Converte Milimetro em Pulsos
	ConversorMilimPul01ResfrSup02: MmConversorPulso;
	///Bloco Converte Milimetro em Pulsos
	ConversorMilimPul02ResfrSup02: MmConversorPulso;
	///Bloco Converte Pulsos em Milimetros
	ConversorPulMilimResfrSup02: PulsoConversorMm;
	PulsoChDutosSup02Po: PulsoPositivo;
	PulsoChDutosSup02Ne: PulsoNegativo;
	xAbreDuctosResfriadorSup02: BOOL;
	xFechaDuctosResfriadorSup02: BOOL;
	xAbreResfridorSup02: BOOL;
	xFechaResfridorSup02: BOOL;
	xAjustarAlturaResfriadorSup02: BOOL;
	///Recebera uma valor fixo
	iVelocidadeHomeDuctosResfrSup02: INT;
	iVelocidadeJogDuctosResfrSup02: INT;
	iVelocidadeDuctosResfriadorSup02: INT;
	dValEncoAltura01ResfriadorSup02: DINT;
	dValEncoAltura02ResfriadorSup02: DINT;
	dValEncoAltura03ResfriadorSup02: DINT;
	dValEncoAlturaResfriadorSup02: DINT;
	dValEncoToleranciaResfrSup02: DINT;
	dValEncoAlturaVelMinimaResfrSup02: DINT := 35;
	xDifusorSup02Fechando: BOOL;
	xDifusorSup02Abrindo: BOOL;
	iCompValAltura01ResfriadorSup02: INT;
	iCompValAltura02ResfriadorSup02: INT;
	iCompValAltura03ResfriadorSup02: INT;
	iCompAlturaAtualDuctosResfriadorSup02: INT;
	iCompessaAlturaDuctosResfriadorSup02: INT;
	xPulsoChDutosSup02Po: BOOL;
	xPulsoChDutosSup02Ne: BOOL;
END_VAR

iCompessaAlturaDuctosResfriadorSup02:=REAL_TO_INT(rOffSetResfSup02);
iCompValAltura01ResfriadorSup02:=	iValAltura01ResfriadorSup02 - iCompessaAlturaDuctosResfriadorSup02;
iCompValAltura02ResfriadorSup02:=	iValAltura02ResfriadorSup02 - iCompessaAlturaDuctosResfriadorSup02;
iCompValAltura03ResfriadorSup02:=	iValAltura03ResfriadorSup02 - iCompessaAlturaDuctosResfriadorSup02;

// CONVERSÃO MILIMETROS EM PULSOS
ConversorMilimPul01ResfrSup02(
	dPulso:= 1051,
	dMilimetro:= 114,
	iEntrMilimetro01:= iCompValAltura01ResfriadorSup02,
	iEntrMilimetro02:= iCompValAltura02ResfriadorSup02,
	iEntrMilimetro03:= iCompValAltura03ResfriadorSup02,
	dSaidaPulso01=> dValEncoAltura01ResfriadorSup02,
	dSaidaPulso02=> dValEncoAltura02ResfriadorSup02,
	dSaidaPulso03=> dValEncoAltura03ResfriadorSup02);

ConversorMilimPul02ResfrSup02(
	dPulso:= 1051,
	dMilimetro:= 114,
	iEntrMilimetro01:= 2,//iValEncoToleranciaDuctosSup02,
	iEntrMilimetro02:= 10,//iValEncoAlturaVelMinimaDuctosSup02,
	dSaidaPulso01=> dValEncoToleranciaResfrSup02,
	dSaidaPulso02=> dValEncoAlturaVelMinimaResfrSup02);

// SEQUENCIA DE HOME

CASE PassoHomeDuctosResfrSup02 OF

		0:	IF xIniciaHomeDuctosSup02 (*OR xAutoHomeResfSup02*) THEN
				PassoHomeDuctosResfrSup02:=5;
			END_IF

		5:	IF xChAbreDuctosResfriadorSup02 THEN
				PassoHomeDuctosResfrSup02:=6;
			ELSE
				PassoHomeDuctosResfrSup02:=10;
			END_IF

		6:	xAutoHomeResfSup02:=FALSE;
			xIniciaHomeDuctosSup02:=FALSE;
			PassoHomeDuctosResfrSup02:=0;

		10:	xIniciaHomeDuctosSup02:=FALSE;
			xHomeDuctosResfriadorSup02Ok:=FALSE;
			xAjusteAlturaDuctosSup02OK:=FALSE;
			xDuctosSup02EmHome:=TRUE;
			iVelocidadeDuctosResfriadorSup02:= 150;//1*iVelocidadeHomeDuctosResfrSup02;
			PassoHomeDuctosResfrSup02:=15;

		15: xFechaResfridorSup02:=TRUE;
			PassoHomeDuctosResfrSup02:=20;

		20:	IF xSensorFechadoResfriadorSup02 THEN
				PassoHomeDuctosResfrSup02:=50;
			END_IF
			IF xPause THEN
				PassoPausaHomeDuctosResfrSup02:=10;
				PassoHomeDuctosResfrSup02:=300;
			END_IF
			IF xAlarmeMotorDifusorSup02 THEN
				PassoAlmHomeDuctosResfrSup02:=10;
				PassoHomeDuctosResfrSup02:=400;
			END_IF

		50:	xFechaResfridorSup02:=FALSE;
			PassoHomeDuctosResfrSup02:=55;

		55:	iVelocidadeDuctosResfriadorSup02:= 50;
			PassoHomeDuctosResfrSup02:=56;

		56:	xAbreResfridorSup02:=TRUE;
			PassoHomeDuctosResfrSup02:=60;

		60:	IF NOT xSensorFechadoResfriadorSup02 THEN
				PassoHomeDuctosResfrSup02:=70;
			END_IF
			IF xPause THEN
				PassoPausaHomeDuctosResfrSup02:=50;
				PassoHomeDuctosResfrSup02:=300;
			END_IF
			IF xAlarmeMotorDifusorSup02 THEN
				PassoAlmHomeDuctosResfrSup02:=50;
				PassoHomeDuctosResfrSup02:=400;
			END_IF

		70:	xAbreResfridorSup02:=FALSE;
			PassoHomeDuctosResfrSup02:=74;

		74:	IF NOT xMotorDifusorSup02Ligado THEN
				PassoHomeDuctosResfrSup02:=75;
			END_IF

		75: xHomeEncoderDuctosResfriadorSup02:=TRUE;
			PassoHomeDuctosResfrSup02:=80;

		80: xHomeEncoderDuctosResfriadorSup02:=FALSE;
			xDuctosSup02EmHome:=FALSE;
			xAutoHomeResfSup02:=FALSE;
			xHomeDuctosResfriadorSup02Ok:=TRUE;
			PassoHomeDuctosResfrSup02:=0;

		// Emergência Pausa/Reinicio
		300:xFechaResfridorSup02:=FALSE;
			xAbreResfridorSup02:=FALSE;
			PassoHomeDuctosResfrSup02:=301;

		301:xDuctosSup02EmHome:=FALSE;
			PassoHomeDuctosResfrSup02:=302;

		302:IF xRestart THEN
				PassoHomeDuctosResfrSup02:=303;
			END_IF

		303:PassoHomeDuctosResfrSup02:=0;//PassoPausaHomeDuctosResfrSup02;

		// Alarme Motor Parada/Reinicio
		400:xFechaResfridorSup02:=FALSE;
			xAbreResfridorSup02:=FALSE;
			PassoHomeDuctosResfrSup02:=401;

		401:PassoHomeDuctosResfrSup02:=402;

		402:IF xRestart AND iCanOpenInverDuctResfrSup02StateOk THEN
				PassoHomeDuctosResfrSup02:=PassoAlmHomeDuctosResfrSup02;
			END_IF
END_CASE

//
IF xTerceiroEstagioResfriador THEN
	dValEncoAlturaResfriadorSup02:=dValEncoAltura03ResfriadorSup02;
ELSIF xSegundoEstagioResfriador THEN
	dValEncoAlturaResfriadorSup02:=dValEncoAltura02ResfriadorSup02;
ELSE
	dValEncoAlturaResfriadorSup02:=dValEncoAltura01ResfriadorSup02;
END_IF

// SEQUENCIA DE FUNCIONAMENTO

IF (xBtRecAjustaAlturaDuctosSup02 OR BtParamDuctosResfriadorSup02 OR (xLigaSegEstagDuctosSup02 AND NOT xChAbreDuctosResfriadorSup02) OR (xLigaTerEstagDuctosSup02 AND NOT xChAbreDuctosResfriadorSup02) OR xReajustaAlturaDuctosSup02) AND xHomeDuctosResfriadorSup02Ok THEN
	xAjustarAlturaResfriadorSup02:=TRUE;
	xBtRecAjustaAlturaDuctosSup02:=FALSE;
	BtParamDuctosResfriadorSup02:=FALSE;
	xLigaSegEstagDuctosSup02:= FALSE;
	xLigaTerEstagDuctosSup02:= FALSE;
	xReajustaAlturaDuctosSup02:=FALSE;
ELSE
	xBtRecAjustaAlturaDuctosSup02:=FALSE;
	BtParamDuctosResfriadorSup02:=FALSE;
	xLigaSegEstagDuctosSup02:= FALSE;
	xLigaTerEstagDuctosSup02:= FALSE;
	xReajustaAlturaDuctosSup02:=FALSE;
END_IF

CASE PassoAjusteDuctosResfSup02 OF

		0:	IF xAjustarAlturaResfriadorSup02 AND NOT xAbreDuctosResfriadorSup02 THEN //AND NOT xChAbreDuctosResfriadorSup02 THEN
				PassoAjusteDuctosResfSup02:=10;
			END_IF

		10:	xAjustarAlturaResfriadorSup02:=FALSE;
			xAjusteAlturaDuctosSup02OK:=FALSE;
			xDuctosSup02EmAjuste:=TRUE;
			IF dValorEncoderDuctosResfriadorSup02<dValEncoAlturaResfriadorSup02-dValEncoToleranciaResfrSup02 THEN
				xDifusorSup02Abrindo:=TRUE;
				PassoAjusteDuctosResfSup02:=20;//Abre
			END_IF
			IF dValorEncoderDuctosResfriadorSup02>dValEncoAlturaResfriadorSup02+dValEncoToleranciaResfrSup02 THEN
				PassoAjusteDuctosResfSup02:=100;//Fecha
				xDifusorSup02Fechando:=TRUE;
			END_IF
			IF dValorEncoderDuctosResfriadorSup02>=dValEncoAlturaResfriadorSup02-dValEncoToleranciaResfrSup02 AND dValorEncoderDuctosResfriadorSup02<=dValEncoAlturaResfriadorSup02+dValEncoToleranciaResfrSup02 THEN
				PassoAjusteDuctosResfSup02:=180;//Não se Move
			END_IF
//Abre
		20:	iVelocidadeDuctosResfriadorSup02:= iVelocidadeAjusteDuctosResfriadorSup02;
			PassoAjusteDuctosResfSup02:=25;

		25:	xAbreResfridorSup02:=TRUE;
			PassoAjusteDuctosResfSup02:=30;

		30:	IF (dValorEncoderDuctosResfriadorSup02>=dValEncoAlturaResfriadorSup02-35(*dValEncoAlturaVelMinimaResfrSup02*)) OR xSensorAbertoResfriadorSup02  THEN
				PassoAjusteDuctosResfSup02:=40;
			END_IF
			IF iVelocidadeDuctosResfriadorSup02<> iVelocidadeAjusteDuctosResfriadorSup02 THEN
				PassoAjusteDuctosResfSup02:=20;
			END_IF
			IF xPause THEN
				PassoPausaAjusteDuctosResfSup02:=20;
				PassoAjusteDuctosResfSup02:=300;
			END_IF
			IF xAlarmeMotorDifusorSup02 THEN
				PassoAlmAjusteDuctosResfSup02:=20;
				PassoAjusteDuctosResfSup02:=400;
			END_IF

		40:	iVelocidadeDuctosResfriadorSup02:= iVelocidadeMinimaDuctosResfriadorSup02;
			PassoAjusteDuctosResfSup02:=50;

		50:	IF (dValorEncoderDuctosResfriadorSup02>=dValEncoAlturaResfriadorSup02) OR xSensorAbertoResfriadorSup02 THEN
				PassoAjusteDuctosResfSup02:=60;
			END_IF
			IF xPause THEN
				PassoPausaAjusteDuctosResfSup02:=40;
				PassoAjusteDuctosResfSup02:=300;
			END_IF
			IF xAlarmeMotorDifusorSup02 THEN
				PassoAlmAjusteDuctosResfSup02:=40;
				PassoAjusteDuctosResfSup02:=400;
			END_IF

		60: xAbreResfridorSup02:=FALSE;
			PassoAjusteDuctosResfSup02:=180;

//Desce
		100:iVelocidadeDuctosResfriadorSup02:= 1*iVelocidadeAjusteDuctosResfriadorSup02;
			PassoAjusteDuctosResfSup02:=105;

		105:xFechaResfridorSup02:=TRUE;
			PassoAjusteDuctosResfSup02:=110;

		110:IF (dValorEncoderDuctosResfriadorSup02 <= dValEncoAlturaResfriadorSup02+35(*dValEncoAlturaVelMinimaResfrSup02*)) OR xSensorFechadoResfriadorSup02 THEN
				PassoAjusteDuctosResfSup02:=120;
			END_IF
			IF iVelocidadeDuctosResfriadorSup02<> 1*iVelocidadeAjusteDuctosResfriadorSup02 THEN
				PassoAjusteDuctosResfSup02:=100;
			END_IF
			IF xPause THEN
				PassoPausaAjusteDuctosResfSup02:=100;
				PassoAjusteDuctosResfSup02:=300;
			END_IF
			IF xAlarmeMotorDifusorSup02 THEN
				PassoAlmAjusteDuctosResfSup02:=100;
				PassoAjusteDuctosResfSup02:=400;
			END_IF

		120:iVelocidadeDuctosResfriadorSup02:= 1*iVelocidadeMinimaDuctosResfriadorSup02;
			PassoAjusteDuctosResfSup02:=130;

		130:IF (dValorEncoderDuctosResfriadorSup02<=dValEncoAlturaResfriadorSup02) OR xSensorFechadoResfriadorSup02 THEN
				PassoAjusteDuctosResfSup02:=140;
			END_IF
			IF iVelocidadeDuctosResfriadorSup02<> 1*iVelocidadeMinimaDuctosResfriadorSup02 THEN
				PassoAjusteDuctosResfSup02:=120;
			END_IF
			IF xPause THEN
				PassoPausaAjusteDuctosResfSup02:=120;
				PassoAjusteDuctosResfSup02:=300;
			END_IF
			IF xAlarmeMotorDifusorSup02 THEN
				PassoAlmAjusteDuctosResfSup02:=120;
				PassoAjusteDuctosResfSup02:=400;
			END_IF

		140:xFechaResfridorSup02:=FALSE;
			PassoAjusteDuctosResfSup02:=180;
//Fim
		180:xDifusorSup02Abrindo:=FALSE;
			xDifusorSup02Fechando:=FALSE;
			xDuctosSup02EmAjuste:=FALSE;
			xAjusteAlturaDuctosSup02OK:=TRUE;
			PassoAjusteDuctosResfSup02:=0;

		// Emergência Pausa/Reinicio
		300:xAbreResfridorSup02:=FALSE;
			xFechaResfridorSup02:=FALSE;
			PassoAjusteDuctosResfSup02:=301;

		301:PassoAjusteDuctosResfSup02:=302;

		302:IF xRestart THEN
				PassoAjusteDuctosResfSup02:=303;
			END_IF

		303:PassoAjusteDuctosResfSup02:=PassoPausaAjusteDuctosResfSup02;

		// Alarme Motor Parada/Reinicio
		400:xAbreResfridorSup02:=FALSE;
			xFechaResfridorSup02:=FALSE;
			PassoAjusteDuctosResfSup02:=401;

		401:PassoAjusteDuctosResfSup02:=402;

		402:IF xRestart AND iCanOpenInverDuctResfrSup02StateOk THEN
				PassoAjusteDuctosResfSup02:=PassoAlmAjusteDuctosResfSup02;
			END_IF

END_CASE

// MOVIMENTO COM A CHAVE DE ABERTURA

PulsoChDutosSup02Po(Entrada:= xChAbreDuctosResfriadorSup02, SaidaPulsoPo=> xPulsoChDutosSup02Po);
PulsoChDutosSup02Ne(Entrada:= xChAbreDuctosResfriadorSup02, SaidaPulsoNe=> xPulsoChDutosSup02Ne);

IF xPulsoChDutosSup02Po THEN
	xPausaMesaResfrimento:=TRUE;
END_IF
IF xPulsoChDutosSup02Ne THEN
	xPausaMesaResfrimento:=FALSE;
END_IF

CASE PassoChaveDuctosResfrSup02 OF

		0:	IF xPulsoChDutosSup02Po AND xHomeDuctosResfriadorSup02Ok THEN //IF xChAbreDuctosResfriadorSup02 AND xHomeDuctosResfriadorSup02Ok THEN
				PassoChaveDuctosResfrSup02:=5;
				PassoAjusteDuctosResfSup02:=0;
				xFechaResfridorSup02:=FALSE;
			END_IF

		5:	IF NOT xPrimeiroEstagioResfriador THEN
				PassoChaveDuctosResfrSup02:=10;
			END_IF

		10:	iVelocidadeDuctosResfriadorSup02:=iVelocidadeAjusteDuctosResfriadorSup02;
			xAjusteAlturaDuctosSup02OK:=FALSE;
			xAbreDuctosResfriadorSup02:=TRUE;//xChAbreDuctosResfriadorSup02;
			IF xSensorAbertoResfriadorSup02 THEN
				PassoChaveDuctosResfrSup02:=20;
			END_IF
			IF xPause THEN
				PassoPausaChaveDuctosResfrSup02:=10;
				PassoChaveDuctosResfrSup02:=300;
			END_IF
			IF xAlarmeMotorDifusorSup02 THEN
				PassoAlmChaveDuctosResfrSup02:=10;
				PassoChaveDuctosResfrSup02:=400;
			END_IF

		20:	xAbreDuctosResfriadorSup02:=FALSE;
			PassoChaveDuctosResfrSup02:=21;

		21:	IF xPulsoChDutosSup02Ne THEN//IF NOT xChAbreDuctosResfriadorSup02 THEN
				xAbreDuctosResfriadorSup02:=FALSE;
				PassoChaveDuctosResfrSup02:=0;
				PassoAjusteDuctosResfSup02:=100;
			END_IF
			IF xPause THEN
				PassoPausaChaveDuctosResfrSup02:=21;
				PassoChaveDuctosResfrSup02:=300;
			END_IF
			IF xAlarmeMotorDifusorSup02 THEN
				PassoAlmChaveDuctosResfrSup02:=21;
				PassoChaveDuctosResfrSup02:=400;
			END_IF

		// Emergência Pausa/Reinicio
		300:xAbreDuctosResfriadorSup02:=FALSE;
			PassoChaveDuctosResfrSup02:=301;

		301:PassoChaveDuctosResfrSup02:=302;

		302:IF xRestart THEN
				PassoChaveDuctosResfrSup02:=303;
			END_IF

		303:PassoChaveDuctosResfrSup02:=PassoPausaChaveDuctosResfrSup02;

		// Alarme Motor Parada/Reinicio
		400:xAbreDuctosResfriadorSup02:=FALSE;
			PassoChaveDuctosResfrSup02:=401;

		401:PassoChaveDuctosResfrSup02:=402;

		402:IF xRestart AND iCanOpenInverDuctResfrSup02StateOk THEN
				PassoChaveDuctosResfrSup02:=PassoAlmChaveDuctosResfrSup02;
			END_IF

END_CASE

// MOVIMENTAÇÃO PELO COMANDO ENTRADAS DIGITAIS DO INVERSOR
// Comando e Dirreção
xMotorResfridorSup02Abre:= xAbreResfridorSup02 OR xAbreDuctosResfriadorSup02;
xMotorResfridorSup02Fecha:= xFechaResfridorSup02;

InversorResfSup02.i_xAvanco:=xMotorResfridorSup02Abre;
InversorResfSup02.i_xRecuo:=xMotorResfridorSup02Fecha;
// Velocidade
InversorResfSup02.i_iFreqRef:=iVelocidadeDuctosResfriadorSup02;
//---------------------------------------------------------------------------------\\

ConversorPulMilimResfrSup02(
	dPulso:= 1051,
	dMilimetro:= 114,
	dEntradaPulso01:= dValorEncoderDuctosResfriadorSup02,
	iSaidaMilimetro01=> iCompAlturaAtualDuctosResfriadorSup02 );

iAlturaAtualDuctosResfriadorSup02:=iCompAlturaAtualDuctosResfriadorSup02+iCompessaAlturaDuctosResfriadorSup02;

IF xOperacaoManual THEN
	PassoHomeDuctosResfrSup02:=0;
	PassoPausaHomeDuctosResfrSup02:=0;
	PassoAlmHomeDuctosResfrSup02:=0;
	PassoAjusteDuctosResfSup02:=0;
	PassoPausaAjusteDuctosResfSup02:=0;
	PassoAlmAjusteDuctosResfSup02:=0;
	PassoChaveDuctosResfrSup02:=0;
	PassoPausaChaveDuctosResfrSup02:=0;
	PassoAlmChaveDuctosResfrSup02:=0;
	xIniciaHomeDuctosSup02:=FALSE;
	xHomeEncoderDuctosResfriadorSup02:=FALSE;
	xAbreDuctosResfriadorSup02:=FALSE;
	xFechaDuctosResfriadorSup02:=FALSE;
	xDifusorSup02Abrindo:=FALSE;
	xDifusorSup02Fechando:=FALSE;
	xAjusteAlturaDuctosSup02OK:=FALSE;
	xFechaDuctosResfriadorSup02:=FALSE;
	xBtRecAjustaAlturaDuctosSup02:=FALSE;
	BtParamDuctosResfriadorSup02:=FALSE;
	xDuctosSup02EmHome:=FALSE;
	xDuctosSup02EmAjuste:=FALSE;
	xLigaSegEstagDuctosSup02:= FALSE;
	xLigaTerEstagDuctosSup02:= FALSE;
	xReajustaAlturaDuctosSup02:=FALSE;
	xDesceAutoFimCiclo:=FALSE;

	xFechaResfridorSup02:=FALSE;
	xAbreResfridorSup02:=FALSE;
	xLigaTerEstagDuctosSup02:=FALSE;
END_IF

(* ---- K_Guilhotina01.prg.st ---- *)
PROGRAM K_Guilhotina01
VAR
	PassoHomeGuilhotina01: INT;
	PassoAjusteGuilhotina01: INT;
	PassoPausaHomeGuilhotina01: INT;
	PassoPausaAjusteGuilhotina01: INT;
	PassoAlmHomeGuilhotina01: INT;
	PassoAlmAjusteGuilhotina01: INT;
	xSinalAjusteG01: INT;
	ContadorEncoderPo: ContadorUpDown;
	TonHomeGuilho01: TON;
	xTonHomeGuilho01In: BOOL;
	xTonHomeGuilho01Q: BOOL;
	///Bloco Converte Milimetro em Pulsos
	ConversorMilimPul01Guilho01: MmConversorPulso;
	///Bloco Converte Milimetro em Pulsos
	ConversorMilimPul02Guilho01: MmConversorPulso;
	///Bloco Converte Pulsos em Milimetros
	ConversorPulMilimGuilho01: PulsoConversorMm;
	xExecutaMovGuilhotina01: BOOL;
	xExecutaStopGuilhotina01: BOOL;
	xStopGuilhotina01Done: BOOL;
	xSetValorSpAltGuil01Sup: BOOL;
	iAlturaGhilhotina01Aux: INT;
	xAjustarAlturaGuilhotina01: BOOL;
	iVelocidadeHomeGuilhotina01: INT;
	iVelocidadeGuilhotina01: INT;
	dValEncoAlturaGuilhotina01: DINT;
	dValEncoToleranciaGuilhotina01: DINT;
	dValEncoAlturaVelMinGuilhotina01: DINT;
	xCmdPositivoGuilhotina01: BOOL;
	xCmdNegativoGuilhotina01: BOOL;
	xIncrementaEncoderGuilhotina01Po: BOOL;
	xDecrementaEncoderGuilhotina01Po: BOOL;
	iValorEncoderGuilhotina01Po: INT;
	xSobeJogGuilhotina01: BOOL;
	xDesceJogGuilhotina01: BOOL;
	xSobeGuilhotina01: BOOL;
	xDesceGuilhotina01: BOOL;
END_VAR

IF iAlturaGhilhotina01 <> iAlturaGhilhotina01Aux THEN
	xSetValorSpAltGuil01Sup:=TRUE;

END_IF;

IF xSetValorSpAltGuil01Sup THEN
	iAlturaGhilhotina01Aux:=iAlturaGhilhotina01;
ELSE
	IF NOT xMotorGuilhotina01Ligado THEN
		iAlturaGhilhotina01:=iAlturaAtualGuilhotina01;
	END_IF;
END_IF

IF iAlturaGhilhotina01Aux=iAlturaAtualGuilhotina01 THEN
	xSetValorSpAltGuil01Sup:=FALSE;
END_IF

// CONVERSÃO MILIMETROS EM PULSOS

ConversorMilimPul01Guilho01(
	dPulso:= 110981,
	dMilimetro:= 100,
	iEntrMilimetro01:= iAlturaGhilhotina01Aux,//iAlturaGhilhotina02,
	dSaidaPulso01=> dValEncoAlturaGuilhotina01);

ConversorMilimPul02Guilho01(
	dPulso:= 110981,
	dMilimetro:= 100,
	iEntrMilimetro01:= 2,//iValEncoToleranciaGuilhotina,
	iEntrMilimetro02:= 8,//iValEncoAlturaVelMinGuilhotina,
	dSaidaPulso01=> dValEncoToleranciaGuilhotina01,
	dSaidaPulso02=> dValEncoAlturaVelMinGuilhotina01);

// SEQUENCIA DE HOME

CASE PassoHomeGuilhotina01 OF

		0:	IF xIniciaHomeGuilhotina01 OR xAutoHomeGuilho01 THEN
				PassoHomeGuilhotina01:=5;
			END_IF

		5:	xIniciaHomeGuilhotina01:=FALSE;
			xAutoHomeGuilho01:=FALSE;
			xGuilhotina01EmAjuste:=FALSE;
			xHomeGuilhotina01Ok:=FALSE;
			xAjusteAlturaGuilhotina01OK:=FALSE;
			xGuilhotina01EmHome:=TRUE;
			PassoHomeGuilhotina01:=8;

		8: IF xSensorZeroGuilhotina01 THEN
				PassoHomeGuilhotina01:=9;
			ELSE
				PassoHomeGuilhotina01:=13;
			END_IF

		9: iVelocidadeGuilhotina01:= 600;//iVelocidadeHomeGuilhotina01;
		   PassoHomeGuilhotina01:=10;

		10:	xSobeGuilhotina01:=TRUE;
			PassoHomeGuilhotina01:=11;

		11: IF NOT xSensorZeroGuilhotina01 THEN
				PassoHomeGuilhotina01:=30;
			END_IF
			IF xPause THEN
				PassoPausaHomeGuilhotina01:=50;
				PassoHomeGuilhotina01:=300;
			END_IF
			IF xAlarmeMotorGuilhotina01 THEN
				PassoAlmHomeGuilhotina01:=50;
				PassoHomeGuilhotina01:=400;
			END_IF

		13:	PassoHomeGuilhotina01:=14;

		14:	iVelocidadeGuilhotina01:= 600;//iVelocidadeHomeGuilhotina01;
			xSinalAjusteG01:=1;
			PassoHomeGuilhotina01:=15;

		15:	xSobeGuilhotina01:=TRUE;
			PassoHomeGuilhotina01:=20;

		20:	IF xSensorPositivoGuilhotina01 THEN
				PassoHomeGuilhotina01:=30;
			END_IF
			IF xSensorZeroGuilhotina01 THEN
				PassoHomeGuilhotina01:=9;//50;
			END_IF
			IF xPause THEN
				PassoPausaHomeGuilhotina01:=15;
				PassoHomeGuilhotina01:=300;
			END_IF
			IF xAlarmeMotorGuilhotina01 THEN
				PassoAlmHomeGuilhotina01:=15;
				PassoHomeGuilhotina01:=400;
			END_IF

		30: xSobeGuilhotina01:=TRUE;
			PassoHomeGuilhotina01:=31;

		31:	iVelocidadeGuilhotina01:=-1*600;//iVelocidadeHomeGuilhotina01;
			xSinalAjusteG01:=-1;
			PassoHomeGuilhotina01:=40;

		40:	IF xSensorNegativoGuilhotina01 THEN
				PassoHomeGuilhotina01:=13;
			END_IF
			IF xSensorZeroGuilhotina01 THEN
				PassoHomeGuilhotina01:=50;
			END_IF
			IF xPause THEN
				PassoPausaHomeGuilhotina01:=30;
				PassoHomeGuilhotina01:=300;
			END_IF
			IF xAlarmeMotorGuilhotina01 THEN
				PassoAlmHomeGuilhotina01:=30;
				PassoHomeGuilhotina01:=400;
			END_IF

		50: iVelocidadeGuilhotina01:= xSinalAjusteG01*150;
			PassoHomeGuilhotina01:=53;

		53:	xTonHomeGuilho01In:=TRUE;
			PassoHomeGuilhotina01:=54;

		54: IF xTonHomeGuilho01Q THEN
				PassoHomeGuilhotina01:=60;
			END_IF

		60:	xTonHomeGuilho01In:=FALSE;
			PassoHomeGuilhotina01:=70;

		70: xSobeGuilhotina01:=FALSE;
			PassoHomeGuilhotina01:=80;

		80: xHomeEncoderGuilhotinaResfriador01:=TRUE;
			PassoHomeGuilhotina01:=81;

		81:PassoHomeGuilhotina01:=82;

		82: xHomeEncoderGuilhotinaResfriador01:=FALSE;
			PassoHomeGuilhotina01:=83;

		83:	xHomeGuilhotina01Ok:=TRUE;
			xGuilhotina01EmHome:=FALSE;
			PassoHomeGuilhotina01:=0;

		// Emergência Pausa/Reinicio
		300:xSobeGuilhotina01:=FALSE;
			xDesceGuilhotina01:=FALSE;
			PassoHomeGuilhotina01:=301;

		301:xGuilhotina01EmHome:=FALSE;
			PassoHomeGuilhotina01:=302;

		302:IF xRestart THEN
				PassoHomeGuilhotina01:=303;
			END_IF

		303:PassoHomeGuilhotina01:=0;//PassoPausaHomeGuilhotina;

		// Alarme Motor Parada/Reinicio
		400:xSobeGuilhotina01:=FALSE;
			xDesceGuilhotina01:=FALSE;
			PassoHomeGuilhotina01:=401;

		401:PassoHomeGuilhotina01:=402;

		402:IF xRestart AND iCanOpenInverGuilResfr01StateOk THEN
				PassoHomeGuilhotina01:=PassoAlmHomeGuilhotina01;
			END_IF

END_CASE

TonHomeGuilho01(IN:= xTonHomeGuilho01In, PT:=T#1720MS , Q=> xTonHomeGuilho01Q, ET=> );

// SEQUENCIA DE FUNCIONAMENTO

IF (xBtRecAjustaGuilhotina01 OR BtParamGuilhotina01) AND xHomeGuilhotina01Ok THEN
	xAjustarAlturaGuilhotina01:=TRUE;
	xBtRecAjustaGuilhotina01:=FALSE;
	BtParamGuilhotina01:=FALSE;
ELSE
	xBtRecAjustaGuilhotina01:=FALSE;
	BtParamGuilhotina01:=FALSE;
END_IF

CASE PassoAjusteGuilhotina01 OF

		0:	IF xAjustarAlturaGuilhotina01 THEN
				PassoAjusteGuilhotina01:=10;
			END_IF

		10:	xAjustarAlturaGuilhotina01:=FALSE;
			xAjusteAlturaGuilhotina01OK:=FALSE;
			xGuilhotina01EmAjuste:=TRUE;
			IF (dValorEncoderGuilhotinaResfriador01>=dValEncoAlturaGuilhotina01-dValEncoToleranciaGuilhotina01) AND (dValorEncoderGuilhotinaResfriador01<=dValEncoAlturaGuilhotina01+dValEncoToleranciaGuilhotina01) THEN
				PassoAjusteGuilhotina01:=180;//Não se Move
			END_IF
			IF dValorEncoderGuilhotinaResfriador01<dValEncoAlturaGuilhotina01-dValEncoToleranciaGuilhotina01 THEN
				PassoAjusteGuilhotina01:=20;//Sobe
			END_IF
			IF dValorEncoderGuilhotinaResfriador01>dValEncoAlturaGuilhotina01+dValEncoToleranciaGuilhotina01 THEN
				PassoAjusteGuilhotina01:=100;//Desce
			END_IF

//Sobe
		20:	iVelocidadeGuilhotina01:= iVelocidadeAjusteGuilhotina01;
			PassoAjusteGuilhotina01:=25;

		25: xSobeGuilhotina01:=TRUE;
			PassoAjusteGuilhotina01:=30;

		30:	IF dValorEncoderGuilhotinaResfriador01>=dValEncoAlturaGuilhotina01-dValEncoAlturaVelMinGuilhotina01 THEN
				PassoAjusteGuilhotina01:=40;
			END_IF
			IF iVelocidadeGuilhotina01<> iVelocidadeAjusteGuilhotina01 THEN
				PassoAjusteGuilhotina01:=20;
			END_IF
			IF xSensorPositivoGuilhotina01 THEN
				PassoAjusteGuilhotina01:=200;
			END_IF

			IF xPause THEN
				PassoPausaAjusteGuilhotina01:=20;
				PassoAjusteGuilhotina01:=300;
			END_IF
			IF xAlarmeMotorGuilhotina01 THEN
				PassoAlmAjusteGuilhotina01:=20;
				PassoAjusteGuilhotina01:=400;
			END_IF

		40:	iVelocidadeGuilhotina01:= iVelocidadeMinimaGuilhotina01;
			PassoAjusteGuilhotina01:=50;

		50:	IF dValorEncoderGuilhotinaResfriador01>=dValEncoAlturaGuilhotina01 THEN
				PassoAjusteGuilhotina01:=60;
			END_IF
			IF iVelocidadeGuilhotina01<> iVelocidadeMinimaGuilhotina01 THEN
				PassoAjusteGuilhotina01:=40;
			END_IF
			IF xPause THEN
				PassoPausaAjusteGuilhotina01:=40;
				PassoAjusteGuilhotina01:=300;
			END_IF
			IF xAlarmeMotorGuilhotina01 THEN
				PassoAlmAjusteGuilhotina01:=40;
				PassoAjusteGuilhotina01:=400;
			END_IF

		60: xSobeGuilhotina01:=FALSE;
			PassoAjusteGuilhotina01:=180;
//Desce

		100:iVelocidadeGuilhotina01:= 1*iVelocidadeAjusteGuilhotina01;
			PassoAjusteGuilhotina01:=105;

		105:xDesceGuilhotina01:=TRUE;
			PassoAjusteGuilhotina01:=110;

		110:IF dValorEncoderGuilhotinaResfriador01<dValEncoAlturaGuilhotina01+dValEncoAlturaVelMinGuilhotina01 THEN
				PassoAjusteGuilhotina01:=120;
			END_IF
			IF iVelocidadeGuilhotina01<> 1*iVelocidadeAjusteGuilhotina01 THEN
				PassoAjusteGuilhotina01:=100;
			END_IF
			IF	xSensorNegativoGuilhotina01 THEN
				PassoAjusteGuilhotina01:=200;
			END_IF
			IF xPause THEN
				PassoPausaAjusteGuilhotina01:=100;
				PassoAjusteGuilhotina01:=300;
			END_IF
			IF xAlarmeMotorGuilhotina01 THEN
				PassoAlmAjusteGuilhotina01:=100;
				PassoAjusteGuilhotina01:=400;
			END_IF

		120:iVelocidadeGuilhotina01:= 1*iVelocidadeMinimaGuilhotina01;
			PassoAjusteGuilhotina01:=130;

		130:IF  dValorEncoderGuilhotinaResfriador01<=dValEncoAlturaGuilhotina01 THEN
				PassoAjusteGuilhotina01:=140;
			END_IF
			IF xPause THEN
				PassoPausaAjusteGuilhotina01:=120;
				PassoAjusteGuilhotina01:=300;
			END_IF
			IF xAlarmeMotorGuilhotina01 THEN
				PassoAlmAjusteGuilhotina01:=120;
				PassoAjusteGuilhotina01:=400;
			END_IF

		140:xDesceGuilhotina01:=FALSE;
			PassoAjusteGuilhotina01:=180;
//Fim
		180:xExecutaStopGuilhotina01:=FALSE;
			xAjusteAlturaGuilhotina01OK:=TRUE;
			xGuilhotina01EmAjuste:=FALSE;
			PassoAjusteGuilhotina01:=0;

		200:xSobeGuilhotina01:=FALSE;
			xDesceGuilhotina01:=FALSE;
			PassoAjusteGuilhotina01:=0;

		// Emergência Pausa/Reinicio
		300:xSobeGuilhotina01:=FALSE;
			xDesceGuilhotina01:=FALSE;
			PassoAjusteGuilhotina01:=301;

		301:PassoAjusteGuilhotina01:=302;

		302:IF xRestart THEN
				PassoAjusteGuilhotina01:=303;
			END_IF

		303: PassoAjusteGuilhotina01:=PassoPausaAjusteGuilhotina01;

		// Alarme Motor Parada/Reinicio
		400:xSobeGuilhotina01:=FALSE;
			xDesceGuilhotina01:=FALSE;
			PassoAjusteGuilhotina01:=401;

		401:PassoAjusteGuilhotina01:=402;

		402:IF xRestart AND iCanOpenInverGuilResfr01StateOk THEN
				PassoAjusteGuilhotina01:=PassoAlmAjusteGuilhotina01;
			END_IF

END_CASE

// MOVIMENTAÇÃO PELO COMANDO ENTRADAS DIGITAIS DO INVERSOR
// Comando e Dirreção
xMotorGuilhotina01Sobe:= xSobeGuilhotina01 OR xSobeJogGuilhotina01;
xMotorGuilhotina01Desce:= xDesceGuilhotina01 OR xDesceJogGuilhotina01;

InversorGuilhot01.i_xAvanco:=xMotorGuilhotina01Sobe;
InversorGuilhot01.i_xRecuo:=xMotorGuilhotina01Desce;

// Velocidade
InversorGuilhot01.i_iFreqRef:=iVelocidadeGuilhotina01;
//---------------------------------------------------------------------------------\\

ConversorPulMilimGuilho01(
	dPulso:=110981,
	dMilimetro:= 100,
	dEntradaPulso01:= dValorEncoderGuilhotinaResfriador01,
	iSaidaMilimetro01=> iAlturaAtualGuilhotina01 );

IF xOperacaoManual THEN
	PassoHomeGuilhotina01:=0;
	PassoAjusteGuilhotina01:=0;
	xIniciaHomeGuilhotina01:=FALSE;
	xAjusteAlturaGuilhotina01OK:=FALSE;
	xGuilhotina01EmHome:=FALSE;
	xGuilhotina01EmAjuste:=FALSE;

	xSobeGuilhotina01:=FALSE;
	xDesceGuilhotina01:=FALSE;
END_IF

(*-------------------- Manual Jog--------------------------*)

xSobeJogGuilhotina01:=xBtSobeGuilhtina01Manual AND NOT xSensorPositivoGuilhotina01 AND NOT xPausaEmergencia ;
xDesceJogGuilhotina01:=xBtDesceGuilhotina01Manual AND NOT xSensorNegativoGuilhotina01 AND NOT xPausaEmergencia ;
